METHOD INTERNAL ParseResponsePayload : DINT
VAR_INPUT
  /// Response data
  ResponseData : RobotLibraryRecvDataFB;
  /// Timestamp
  Timestamp    : SystemTime;  
END_VAR
// Table 6-77: Received CMD payload (RC to PLC) of "SwitchLanguage"
// --------------------------
// Header
// --------------------------
// Byte 00 : USINT - ParSeq | State     
// Byte 01 : SINT  - AlarmMessageSeverity    
// Byte 02 : UINT  - AlarmMessageCode HB
// Byte 03 :       - AlarmMessageCode LB
// --------------------------
// Datablock
// --------------------------
// Byte 04  : BOOL - SoftMovement
// call base implementation to parse the header from payload buffer
ResponseData.PayloadPtr := SUPER^.ParseResponsePayload(ResponseData := ResponseData, Timestamp := Timestamp);

// copy parsed header to response
_response.ParSeq               := _rspHeader.ParSeq;
_response.State                := _rspHeader.State;
_response.AlarmMessageSeverity := _rspHeader.AlarmMessageSeverity;
_response.AlarmMessageCode     := _rspHeader.AlarmMessageCode;

// Get Response.ActualLanguageCode
_response.ActualLanguageCode := ResponseData.GetString(2);

// Create logging
ParseResponsePayloadLog(ResponseData := ResponseData, Timestamp := Timestamp);
END_METHOD

METHOD INTERNAL ParseResponsePayloadLog
VAR_INPUT
  /// Response data
  ResponseData : RobotLibraryRecvDataFB;
  /// Timestamp
  Timestamp    : SystemTime;  
END_VAR
// Create log entry for Parameter start
CreateLogMessage      ( Timestamp   := Timestamp,
                        MessageType := MessageType.CMD,
                        Severity    := Severity.DEBUG,
                        MessageCode := 0,
                        MessageText := 'Parsed the following parameter(s) from response data:');
                        
// Create log entry for ActualLanguageCode
CreateLogMessagePara1 ( Timestamp   := Timestamp,
                        MessageType := MessageType.CMD,
                        Severity    := Severity.DEBUG,
                        MessageCode := 0,
                        MessageText := 'Response.ActualLanguageCode = {1}',
                        Para1       := _response.ActualLanguageCode);
END_METHOD

METHOD PROTECTED Reset : DINT
VAR_INPUT
END_VAR
Reset := SUPER^.Reset();

Done               := FALSE;
Busy               := FALSE;
CommandBuffered    := FALSE;
END_METHOD

END_FUNCTION_BLOCK

// Library/POUs/General/MC_UserLogin/MC_UserLoginFB
/// Login on RC from PLC
FUNCTION_BLOCK MC_UserLoginFB EXTENDS RobotLibraryBaseExecuteFB
// ------------------------------------------------------------------------- 
//  SRCI Robot Library                                                
// ------------------------------------------------------------------------- 
//                                                                           
//  Object:      UserLoginFB                                       
//  Author:      Thorsten Brach                                                
//  Date:        2024-06-01
//
//  Description:                                              
//   
//                                                                           
//  Copyright: 
//    (C) 2024 Thorsten Brach. All rights reserved                                                                                                                                            
//             Licensed under the LGPL-3.0 license.
//                                                                           
//  Disclaimer:                                                                           
//    This project is provided without any guarantee and can be used for   
//    private and commercial purposes. Any use is at the user’s 
//    own risk and responsibility.
//
// -------------------------------------------------------------------------
VAR_INPUT
  /// Command parameter 
  ParCmd          : UserLoginParCmd;      
END_VAR
VAR_OUTPUT
  /// Command is transferred and confirmed by the RC
  CommandBuffered : BOOL;
  /// command results
  OutCmd          : UserLoginOutCmd;     
END_VAR

VAR
  /// internal copy of command parameter 
 _parCmd          : UserLoginParCmd;
  /// command data to send
 _command         : UserLoginSendData;
  /// response data received
 _response        : UserLoginRecvData;      
END_VAR

SUPER^(AxesGroup := AxesGroup);

METHOD PROTECTED CheckFunctionSupported : BOOL
VAR_IN_OUT
  /// Robot assignment of function
  AxesGroup : AxesGroup; 
END_VAR
CheckFunctionSupported := AxesGroup.InternalData.RCSupportedFunctions.UserLogin;

IF ( NOT CheckFunctionSupported )
THEN
  // call base implementation for set error and create log entry
  SUPER^.CheckFunctionSupported(AxesGroup := AxesGroup);
END_IF
END_METHOD

METHOD PROTECTED CheckParameterChanged : BOOL
VAR_IN_OUT
  /// Robot assignment of function
  AxesGroup    : AxesGroup; 
END_VAR
// Check ParCmd Size is > 0, because MemCmp does not work correctly with size = 0
IF (SIZEOF(ParCmd) = 0) 
THEN 
  RETURN;
END_IF

// compare memory 
_parameterChanged := ( SysDepMemCmp(pData1 := ADR(ParCmd), pData2 := ADR(_parCmd), DataLen := SIZEOF(ParCmd)) <> RobotLibraryConstants.OK );

// check parameter valid ?
_parameterValid   := CheckParameterValid( AxesGroup := AxesGroup );

IF ((  _parameterChanged        )  AND 
    (  _parameterValid          )) OR
    (  _parameterUpdateInternal )  
THEN  
  // reset internal flag for send parameter update
 _parameterUpdateInternal := FALSE;
  // update internal copy of parameters 
 _parCmd := ParCmd;
  // inc parameter sequence
 _command.ParSeq := _command.ParSeq + 1;
  // update command data  
  CommandData := CreateCommandPayload(AxesGroup := AxesGroup); // ( Access via reference to rCommandFB in ACR )
  // notify active command register 
  AxesGroup.Acyclic.ActiveCommandRegister.NotifyParameterChanged := _uniqueID;
END_IF
END_METHOD

METHOD INTERNAL CreateCommandPayload : RobotLibrarySendDataFB
VAR_IN_OUT
  /// Robot assignment of function
  AxesGroup : AxesGroup; 
END_VAR
// Table 6-69: Sent CMD payload (PLC to RC) of "UserLogin"
// --------------------------
// Header
// --------------------------
// Byte 00 : UINT  - Type HB     
// Byte 01 :       - Type LB    
// Byte 02 : USINT - Reserve | ExecutionMode
// Byte 03 : USINT - ParSeq  | Priority
// --------------------------
// Datablock
// --------------------------
// Byte 04 : SINT       - Mode
// Byte 05 : SINT       - LevelID
// Byte 06 : String(50) - Password[0]
// Byte 07 :            - Password[1]
// Byte 08 :            - Password[2]
// Byte 09 :            - Password[3]
// Byte 10 :            - Password[4]
// Byte 11 :            - Password[5]
// Byte 12 :            - Password[6]
// Byte 13 :            - Password[7]
// Byte 14 :            - Password[8]
// Byte 15 :            - Password[9]
// Byte 16 :            - Password[10]
// Byte 17 :            - Password[11]
// Byte 18 :            - Password[12]
// Byte 19 :            - Password[13]
// Byte 20 :            - Password[14]
// Byte 21 :            - Password[15]
// Byte 22 :            - Password[16]
// Byte 23 :            - Password[17]
// Byte 24 :            - Password[18]
// Byte 25 :            - Password[19]
// Byte 26 :            - Password[20]
// Byte 27 :            - Password[21]
// Byte 28 :            - Password[22]
// Byte 29 :            - Password[23]
// Byte 30 :            - Password[24]
// Byte 31 :            - Password[25]
// Byte 32 :            - Password[26]
// Byte 33 :            - Password[27]
// Byte 34 :            - Password[28]
// Byte 35 :            - Password[29]
// Byte 36 :            - Password[30]
// Byte 37 :            - Password[31]
// Byte 38 :            - Password[32]
// Byte 39 :            - Password[33]
// Byte 40 :            - Password[34]
// Byte 41 :            - Password[35]
// Byte 42 :            - Password[36]
// Byte 43 :            - Password[37]
// Byte 44 :            - Password[38]
// Byte 45 :            - Password[39]
// Byte 46 :            - Password[40]
// Byte 47 :            - Password[41]
// Byte 48 :            - Password[42]
// Byte 49 :            - Password[43]
// Byte 50 :            - Password[44]
// Byte 51 :            - Password[45]
// Byte 52 :            - Password[46]
// Byte 53 :            - Password[47]
// Byte 54 :            - Password[48]
// Byte 55 :            - Password[49]
// Byte 56 : String(50) - Username[0]
// Byte 57 :            - Username[1]
// Byte 58 :            - Username[2]
// Byte 59 :            - Username[3]
// Byte 60 :            - Username[4]
// Byte 61 :            - Username[5]
// Byte 62 :            - Username[6]
// Byte 63 :            - Username[7]
// Byte 64 :            - Username[8]
// Byte 65 :            - Username[9]
// Byte 66 :            - Username[10]
// Byte 67 :            - Username[11]
// Byte 68 :            - Username[12]
// Byte 69 :            - Username[13]
// Byte 70 :            - Username[14]
// Byte 71 :            - Username[15]
// Byte 72 :            - Username[16]
// Byte 73 :            - Username[17]
// Byte 74 :            - Username[18]
// Byte 75 :            - Username[19]
// Byte 76 :            - Username[20]
// Byte 77 :            - Username[21]
// Byte 78 :            - Username[22]
// Byte 79 :            - Username[23]
// Byte 80 :            - Username[24]
// Byte 81 :            - Username[25]
// Byte 82 :            - Username[26]
// Byte 83 :            - Username[27]
// Byte 84 :            - Username[28]
// Byte 85 :            - Username[29]
// Byte 86 :            - Username[30]
// Byte 87 :            - Username[31]
// Byte 88 :            - Username[32]
// Byte 89 :            - Username[33]
// Byte 90 :            - Username[34]
// Byte 91 :            - Username[35]
// Byte 92 :            - Username[36]
// Byte 93 :            - Username[37]
// Byte 94 :            - Username[38]
// Byte 95 :            - Username[39]
// Byte 96 :            - Username[40]
// Byte 97 :            - Username[41]
// Byte 98 :            - Username[42]
// Byte 99 :            - Username[43]
// Byte 100:            - Username[44]
// Byte 101:            - Username[45]
// Byte 102:            - Username[46]
// Byte 103:            - Username[47]
// Byte 104:            - Username[48]
// Byte 105:            - Username[49]
// set command parameter 
_command.CmdTyp     :=  CmdType.UserLogin;
_command.ExecMode   :=  ExecMode;
_command.ParSeq     := _command.ParSeq;
_command.Priority   :=  Priority;

_command.Mode       := _parCmd.Mode;
_command.LevelID    := _parCmd.LevelID;
_command.Username   := _parCmd.Username;
_command.Password   := _parCmd.Password;


// copy command data to header
_cmdHeader := _command;
// call base implementation to copy header to payload buffer
CreateCommandPayload := SUPER^.CreateCommandPayload(AxesGroup := AxesGroup);

// add command.Mode
CreateCommandPayload.AddSint(_command.Mode);
// add command.LevelID
CreateCommandPayload.AddSint(_command.LevelID);
// add command.Password
CreateCommandPayload.AddString(_command.Password);
// add command.Username
CreateCommandPayload.AddString(_command.Username);

// Create logging
CreateCommandPayloadLog(AxesGroup := AxesGroup);
END_METHOD

METHOD INTERNAL CreateCommandPayloadLog 
VAR_IN_OUT
  /// Robot assignment of function
  AxesGroup : AxesGroup; 
END_VAR
// Create log entry for Parameter start
CreateLogMessage      ( Timestamp   := AxesGroup.InternalData.SystemTime,
                        MessageType := MessageType.CMD,
                        Severity    := Severity.DEBUG,
                        MessageCode := 0,
                        MessageText := 'Create command payload with the following parameter(s) :');

// Create log entry for Mode
CreateLogMessagePara1 ( Timestamp   := AxesGroup.InternalData.SystemTime,
                        MessageType := MessageType.CMD,
                        Severity    := Severity.DEBUG,
                        MessageCode := 0,
                        MessageText := 'Command.Mode = {1}',
                        Para1       :=  LOGON_MODE_TO_STRING(_command.Mode));

// Create log entry for LevelID
CreateLogMessagePara1 ( Timestamp   := AxesGroup.InternalData.SystemTime,
                        MessageType := MessageType.CMD,
                        Severity    := Severity.DEBUG,
                        MessageCode := 0,
                        MessageText := 'Command.LevelID = {1}',
                        Para1       :=  SINT_TO_STRING(_command.LevelID));

// Create log entry for Password
CreateLogMessagePara1 ( Timestamp   := AxesGroup.InternalData.SystemTime,
                        MessageType := MessageType.CMD,
                        Severity    := Severity.DEBUG,
                        MessageCode := 0,
                        MessageText := 'Command.Password = {1}',
                        Para1       :=  _command.Password);

// Create log entry for Username
CreateLogMessagePara1 ( Timestamp   := AxesGroup.InternalData.SystemTime,
                        MessageType := MessageType.CMD,
                        Severity    := Severity.DEBUG,
                        MessageCode := 0,
                        MessageText := 'Command.Username = {1}',
                        Para1       :=  _command.Username);
END_METHOD

METHOD FB_init : BOOL
VAR_INPUT
  /// if TRUE, the retain variables are initialized (warm start / cold start)
  bInitRetains : BOOL; 
  /// if TRUE, the instance afterwards gets moved into the copy code (online change)
  bInCopyCode  : BOOL;  
END_VAR
MyType := 'MC_UserLoginFB';

ExecMode := ExecutionMode.PARALLEL;
END_METHOD

METHOD PROTECTED OnCall
VAR_IN_OUT
  /// Robot assignment of function
  AxesGroup : AxesGroup; 
END_VAR
// call base implementation
SUPER^.OnCall(AxesGroup := AxesGroup);

CASE _stepCmd OF
  
  00:  IF ( _execute_R.Q )  
       THEN
         // Check function is supported and parameter are valid ?
         IF (( CheckFunctionSupported( AxesGroup := AxesGroup )) AND
             ( CheckParameterValid   ( AxesGroup := AxesGroup )))      
         THEN
           // set busy flag
           Busy := TRUE;
           // Reset command outputs
           SysDepMemSet(pDest := ADR(OutCmd), Value := 0, DataLen := SIZEOF(OutCmd));         
           // apply command parameter
          _parCmd := ParCmd;
           // init parameter sequence
          _command.ParSeq := 1;
           // create command data
           CommandData := CreateCommandPayload(AxesGroup := AxesGroup);
           // Add command to active command register
          _uniqueID := AxesGroup.Acyclic.ActiveCommandRegister.AddCmd( pCommandFB := ADR(THIS^ ));     
           // set timeout
           SetTimeout(PT := _timeoutCmd, rTimer := _timerCmd);
           // inc step counter
          _stepCmd := _stepCmd + 1; 
         END_IF
       END_IF
     

  01:  // Wait for responce received
       IF ( _responseReceived )
       THEN
         // reset response received flag
        _responseReceived := FALSE;

         CASE  _response.State 
         OF
           CmdMessageState.BUFFERED : CommandBuffered := TRUE;
           CmdMessageState.DONE     : Done            := TRUE;
           CmdMessageState.ERROR    : Error           := TRUE;
         END_CASE
                
         // Done, Aborted or Error ?
         IF (_response.State >= CmdMessageState.DONE )
         THEN
           // Reset Busy flag
           Busy := FALSE;
           // Update results
           // set timeout
           SetTimeout(PT := _timeoutCmd, rTimer := _timerCmd);
           // inc step counter
          _stepCmd := _stepCmd + 1; 
         END_IF
       END_IF


  02: IF ( NOT Execute)
      THEN
        Reset();
      END_IF     

ELSE
  // invalid step
  ErrorID := RobotLibraryEvents.ERR_INVALID_STEP;
END_CASE


// Reset FB
IF ( NOT Execute )
THEN
  Reset();
END_IF
END_METHOD

METHOD INTERNAL ParseResponsePayload : DINT
VAR_INPUT
  /// Response data
  ResponseData : RobotLibraryRecvDataFB;
  /// Timestamp
  Timestamp    : SystemTime;  
END_VAR
// Table 6-70: Received CMD payload (RC to PLC) of "UserLogin"
// --------------------------
// Header
// --------------------------
// Byte 00 : USINT - ParSeq | State     
// Byte 01 : SINT  - AlarmMessageSeverity    
// Byte 02 : UINT  - AlarmMessageCode HB
// Byte 03 :       - AlarmMessageCode LB
// --------------------------
// call base implementation to parse the header from payload buffer
ResponseData.PayloadPtr := SUPER^.ParseResponsePayload(ResponseData := ResponseData, Timestamp := Timestamp);

// copy parsed header to response
_response.ParSeq               := _rspHeader.ParSeq;
_response.State                := _rspHeader.State;
_response.AlarmMessageSeverity := _rspHeader.AlarmMessageSeverity;
_response.AlarmMessageCode     := _rspHeader.AlarmMessageCode;

// Create logging
ParseResponsePayloadLog(ResponseData := ResponseData, Timestamp := Timestamp);
END_METHOD

METHOD INTERNAL ParseResponsePayloadLog
VAR_INPUT
  /// Response data
  ResponseData : RobotLibraryRecvDataFB;
  /// Timestamp
  Timestamp    : SystemTime;  
END_VAR
// Create log entry for Parameter start
CreateLogMessage      ( Timestamp   := Timestamp,
                        MessageType := MessageType.CMD,
                        Severity    := Severity.DEBUG,
                        MessageCode := 0,
                        MessageText := 'Parsed the following parameter(s) from response data:');
                        
// Create log entry for no parameter 
CreateLogMessage      ( Timestamp   := Timestamp,
                        MessageType := MessageType.CMD,
                        Severity    := Severity.DEBUG,
                        MessageCode := 0,
                        MessageText := 'This command has no parameter to parse...');
END_METHOD

METHOD PROTECTED Reset : DINT
VAR_INPUT
END_VAR
Reset := SUPER^.Reset();

Done               := FALSE;
Busy               := FALSE;
CommandBuffered    := FALSE;
END_METHOD

END_FUNCTION_BLOCK

// Library/POUs/Read/MC_ReadActualPosition/MC_ReadActualPositionFB
/// Read the actual position – TCP: X…RZ + config/Turn, … Joint: (J1…E6)
FUNCTION_BLOCK MC_ReadActualPositionFB EXTENDS RobotLibraryBaseExecuteFB
// ------------------------------------------------------------------------- 
//  SRCI Robot Library                                                
// ------------------------------------------------------------------------- 
//                                                                           
//  Object:      ReadActualPositionFB                                       
//  Author:      Thorsten Brach                                                
//  Date:        2024-06-01
//
//  Description:                                              
//   
//                                                                           
//  Copyright: 
//    (C) 2024 Thorsten Brach. All rights reserved                                                                                                                                            
//             Licensed under the LGPL-3.0 license.
//                                                                           
//  Disclaimer:                                                                           
//    This project is provided without any guarantee and can be used for   
//    private and commercial purposes. Any use is at the user’s 
//    own risk and responsibility.
//
// -------------------------------------------------------------------------
VAR_INPUT
  /// Processing mode - For more information see chapter 5.6.4.5.
  ProcessingMode     : ProcessingMode;
  /// Defines the target sequence in which the command will be executed
  SequenceFlag       : SequenceFlag;  
  /// command parameter 
  ParCmd             : ReadActualPositionParCmd;
END_VAR

VAR_OUTPUT
  /// TRUE, while the following outputs return valid values
  /// • ActualCartesianPosition
  /// • ToolNoReturn
  /// • FrameNoReturn
  /// • ActualJointPosition
  Valid              : BOOL;
  /// Command is transferred and confirmed by the RC
  CommandBuffered    : BOOL;  
  /// The command was aborted by another command.
  CommandAborted     : BOOL;
  /// TRUE, while command is interrupted during execution and can be continued.
  CommandInterrupted : BOOL;
  /// Receiving of input parameter values has been acknowledged by RC
  ParameterAccepted  : BOOL;
  /// command outputs
  OutCmd             : ReadActualPositionOutCmd;       
END_VAR

VAR
  /// internal copy of command parameter 
 _parCmd             : ReadActualPositionParCmd;
  /// command data to send
 _command            : ReadActualPositionSendData;
  /// response data received
 _response           : ReadActualPositionRecvData;      
END_VAR

SUPER^(AxesGroup := AxesGroup);

METHOD PROTECTED CheckFunctionSupported : BOOL
VAR_IN_OUT
  /// Robot assignment of function
  AxesGroup : AxesGroup; 
END_VAR
CheckFunctionSupported := AxesGroup.InternalData.RCSupportedFunctions.ReadActualPosition;

IF ( NOT CheckFunctionSupported )
THEN
  // call base implementation for set error and create log entry
  SUPER^.CheckFunctionSupported(AxesGroup := AxesGroup);
END_IF
END_METHOD

METHOD PROTECTED CheckParameterChanged : BOOL
VAR_IN_OUT
  /// Robot assignment of function
  AxesGroup    : AxesGroup; 
END_VAR
// Check ParCmd Size is > 0, because MemCmp does not work correctly with size = 0
IF (SIZEOF(ParCmd) = 0) 
THEN 
  RETURN;
END_IF

// compare memory 
_parameterChanged := ( SysDepMemCmp(pData1 := ADR(ParCmd), pData2 := ADR(_parCmd), DataLen := SIZEOF(ParCmd)) <> RobotLibraryConstants.OK );

// check parameter valid ?
_parameterValid   := CheckParameterValid( AxesGroup := AxesGroup );

IF ((  _parameterChanged        )  AND 
    (  _parameterValid          )) OR
    (  _parameterUpdateInternal )  
THEN  
  // reset internal flag for send parameter update
 _parameterUpdateInternal := FALSE;
  // update internal copy of parameters 
 _parCmd := ParCmd;
  // inc parameter sequence
 _command.ParSeq := _command.ParSeq + 1;
  // update command data  
  CommandData := CreateCommandPayload(AxesGroup := AxesGroup); // ( Access via reference to rCommandFB in ACR )
  // notify active command register 
  AxesGroup.Acyclic.ActiveCommandRegister.NotifyParameterChanged := _uniqueID;
  // Reset parameter accepted flag
  ParameterAccepted := FALSE;  
END_IF
END_METHOD

METHOD INTERNAL CreateCommandPayload : RobotLibrarySendDataFB
VAR_IN_OUT
  /// Robot assignment of function
  AxesGroup : AxesGroup; 
END_VAR
// Table 6-38: Sent CMD payload (PLC to RC) of "ReadActualPosition"
// --------------------------
// Header
// --------------------------
// Byte 00 : UINT  - Type HB     
// Byte 01 :       - Type LB    
// Byte 02 : USINT - Reserve | ExecutionMode
// Byte 03 : USINT - ParSeq  | Priority
// --------------------------
// Datablock
// --------------------------
// Byte 04 : SINT  EmitterID[0];
// Byte 05 : SINT  EmitterID[1];
// Byte 06 : SINT  EmitterID[2];
// Byte 07 : SINT  EmitterID[3];
// Byte 08 : SINT  ListenerID;
// Byte 09 : BYTE  Reserved;
// Byte 10 : USINT ToolNo
// Byte 11 : USINT FrameNo
// --------------------------
// set command parameter 
_command.CmdTyp       :=  CmdType.ReadActualPosition;
_command.ExecMode     :=  ExecMode;
_command.ParSeq       := _command.ParSeq;
_command.Priority     :=  Priority;
_command.EmitterID[0] := 0;
_command.EmitterID[1] := 0;
_command.EmitterID[2] := 0;
_command.EmitterID[3] := 0;
_command.Reserve      := 0;
_command.ListenerID   := _parCmd.ListenerID;
_command.ToolNo       := INT_TO_USINT(_parCmd.ToolNo);
_command.FrameNo      := INT_TO_USINT(_parCmd.FrameNo);


// copy command data to header
_cmdHeader := _command;
// call base implementation to copy header to payload buffer
CreateCommandPayload := SUPER^.CreateCommandPayload(AxesGroup := AxesGroup);

// add command.EmitterID[0]
CreateCommandPayload.AddSint(_command.EmitterID[0]);
// add command.EmitterID[1]
CreateCommandPayload.AddSint(_command.EmitterID[1]);
// add command.EmitterID[2]
CreateCommandPayload.AddSint(_command.EmitterID[2]);
// add command.EmitterID[3]
CreateCommandPayload.AddSint(_command.EmitterID[3]);
// add command.ListenerID
CreateCommandPayload.AddSint(_command.ListenerID);
// add command.Reserve
CreateCommandPayload.AddByte(_command.Reserve);
// add command.Index[0]
CreateCommandPayload.AddUsint(_command.ToolNo);
// add command.Index[1]
CreateCommandPayload.AddUsint(_command.FrameNo);

// Create logging
CreateCommandPayloadLog(AxesGroup := AxesGroup);
END_METHOD

METHOD INTERNAL CreateCommandPayloadLog
VAR_IN_OUT
  /// Robot assignment of function
  AxesGroup : AxesGroup; 
END_VAR
VAR 
  /// internal index for loops
 _idx : DINT;
END_VAR
// Create log entry for Parameter start
CreateLogMessage      ( Timestamp   := AxesGroup.InternalData.SystemTime,
                        MessageType := MessageType.CMD,
                        Severity    := Severity.DEBUG,
                        MessageCode := 0,
                        MessageText := 'Create command payload with the following parameter(s) :');
  
// Create log entry for EmitterID[x]
FOR _idx := 0 TO 3
DO
  CreateLogMessagePara2 ( Timestamp   := AxesGroup.InternalData.SystemTime,
                          MessageType := MessageType.CMD,
                          Severity    := Severity.DEBUG,
                          MessageCode := 0,
                          MessageText := 'Command.EmitterID[{2}] = {1}',
                          Para1       :=  SINT_TO_STRING(_command.EmitterID[_idx]),
                          Para2       :=  DINT_TO_STRING(_idx));
END_FOR

// Create log entry for ListenerID
CreateLogMessagePara1 ( Timestamp   := AxesGroup.InternalData.SystemTime,
                        MessageType := MessageType.CMD,
                        Severity    := Severity.DEBUG,
                        MessageCode := 0,
                        MessageText := 'Command.ListenerID = {1}',
                        Para1       :=  SINT_TO_STRING(_command.ListenerID));
                        
// Create log entry for Reserve
CreateLogMessagePara1 ( Timestamp   := AxesGroup.InternalData.SystemTime,
                        MessageType := MessageType.CMD,
                        Severity    := Severity.DEBUG,
                        MessageCode := 0,
                        MessageText := 'Command.Reserve = {1}',
                        Para1       :=  BYTE_TO_STRING(_command.Reserve));

// Create log entry for ToolNo
CreateLogMessagePara1 ( Timestamp   := AxesGroup.InternalData.SystemTime,
                        MessageType := MessageType.CMD,
                        Severity    := Severity.DEBUG,
                        MessageCode := 0,
                        MessageText := 'Command.ToolNo = {1}',
                        Para1       :=  USINT_TO_STRING(_command.ToolNo));

// Create log entry for FrameNo
CreateLogMessagePara1 ( Timestamp   := AxesGroup.InternalData.SystemTime,
                        MessageType := MessageType.CMD,
                        Severity    := Severity.DEBUG,
                        MessageCode := 0,
                        MessageText := 'Command.FrameNo = {1}',
                        Para1       :=  USINT_TO_STRING(_command.FrameNo));
END_METHOD

METHOD FB_init : BOOL
VAR_INPUT
  /// if TRUE, the retain variables are initialized (warm start / cold start)
  bInitRetains : BOOL; 
  /// if TRUE, the instance afterwards gets moved into the copy code (online change)
  bInCopyCode  : BOOL;  
END_VAR
MyType := 'MC_ReadActualPositionFB';

ExecMode := ExecutionMode.PARALLEL;
END_METHOD

METHOD PROTECTED OnCall
VAR_IN_OUT
  /// Robot assignment of function
  AxesGroup : AxesGroup; 
END_VAR
// call base implementation
SUPER^.OnCall(AxesGroup := AxesGroup);

CASE _stepCmd OF
  
  00:  IF ( _execute_R.Q )  
       THEN
         // Check function is supported and parameter are valid ?
         IF (( CheckFunctionSupported( AxesGroup := AxesGroup )) AND
             ( CheckParameterValid   ( AxesGroup := AxesGroup )))      
         THEN
           // set busy flag
           Busy := TRUE;
           // Reset command outputs
           SysDepMemSet(pDest := ADR(OutCmd), Value := 0, DataLen := SIZEOF(OutCmd));         
           // apply command parameter
          _parCmd := ParCmd;
           // init parameter sequence
          _command.ParSeq := 1;
           // create command data
           CommandData := CreateCommandPayload(AxesGroup := AxesGroup);
           // Add command to active command register
          _uniqueID := AxesGroup.Acyclic.ActiveCommandRegister.AddCmd( pCommandFB := ADR(THIS^ ));     
           // set timeout
           SetTimeout(PT := _timeoutCmd, rTimer := _timerCmd);
           // inc step counter
          _stepCmd := _stepCmd + 1;
         END_IF 
       END_IF
     

  01:  // Wait for responce received
       IF ( _responseReceived )
       THEN
         // reset response received flag
        _responseReceived := FALSE;

         CASE  _response.State 
         OF
           CmdMessageState.BUFFERED    : CommandBuffered    := TRUE;
           CmdMessageState.ACTIVE      : ParameterAccepted  := TRUE;           
           CmdMessageState.INTERRUPTED : CommandInterrupted := TRUE;           
           CmdMessageState.DONE        : Done               := TRUE;
           CmdMessageState.ABORTED     : CommandAborted     := TRUE;
           CmdMessageState.ERROR       : Error              := TRUE;
         END_CASE
                
         // Done, Aborted or Error ?
         IF (_response.State >= CmdMessageState.DONE )
         THEN
           // Reset Busy flag
           Busy := FALSE;
           // Update results
           OutCmd.OriginID                := _response.OriginID;
           OutCmd.InvocationCounter       := _response.InvocationCounter;
           OutCmd.ToolNoReturn            := _response.ToolNoReturn;
           OutCmd.FrameNoReturn           := _response.FrameNoReturn;
           OutCmd.ActualCartesianPosition := _response.ActualCartesianPosition;
           OutCmd.ActualJointPosition     := _response.ActualJointPosition;
           // set timeout
           SetTimeout(PT := _timeoutCmd, rTimer := _timerCmd);
           // inc step counter
          _stepCmd := _stepCmd + 1; 
         END_IF
       END_IF


  02: IF ( NOT Execute)
      THEN
        Reset();
      END_IF     
      
ELSE
  // invalid step
  ErrorID := RobotLibraryEvents.ERR_INVALID_STEP;
END_CASE


// Reset FB
IF ( NOT Execute )
THEN
  Reset();
END_IF
END_METHOD

METHOD INTERNAL ParseResponsePayload : DINT
VAR_INPUT
  /// Response data
  ResponseData : RobotLibraryRecvDataFB;
  /// Timestamp
  Timestamp    : SystemTime;  
END_VAR
// Table 6-39: Received CMD payload (RC to PLC) of "ReadActualPosition"
// --------------------------
// Header
// --------------------------
// Byte 00 : USINT   - ParSeq | State     
// Byte 01 : SINT    - AlarmMessageSeverity    
// Byte 02 : UINT    - AlarmMessageCode HB
// Byte 03 :         - AlarmMessageCode LB
// --------------------------
// Datablock
// --------------------------
// Byte 04 : USINT   - InvocationCounter;
// Byte 05 : SINT    - Reserved;
// Byte 06 : INT     - OriginID HW HB;
// Byte 07 :         - OriginID HW LB;
// Byte 08 : USINT   - ToolNoReturn;
// Byte 09 : USINT   - FrameNoReturn;
// Byte 10 : REAL    - ActualCartesianPosition.X HW HB;
// Byte 11 :         - ActualCartesianPosition.X HW LB;
// Byte 12 :         - ActualCartesianPosition.X LW HB;
// Byte 13 :         - ActualCartesianPosition.X LW LB;
// Byte 14 : REAL    - ActualCartesianPosition.Y HW HB;
// Byte 15 :         - ActualCartesianPosition.Y HW LB;
// Byte 16 :         - ActualCartesianPosition.Y LW HB;
// Byte 17 :         - ActualCartesianPosition.Y LW LB;
// Byte 18 : REAL    - ActualCartesianPosition.Z HW HB;
// Byte 19 :         - ActualCartesianPosition.Z HW LB;
// Byte 20 :         - ActualCartesianPosition.Z LW HB;
// Byte 21 :         - ActualCartesianPosition.Z LW LB;
// Byte 22 : REAL    - ActualCartesianPosition.RX HW HB;
// Byte 23 :         - ActualCartesianPosition.RX HW LB;
// Byte 24 :         - ActualCartesianPosition.RX LW HB;
// Byte 25 :         - ActualCartesianPosition.RX LW LB;
// Byte 26 : REAL    - ActualCartesianPosition.RY HW HB;
// Byte 27 :         - ActualCartesianPosition.RY HW LB;
// Byte 28 :         - ActualCartesianPosition.RY LW HB;
// Byte 29 :         - ActualCartesianPosition.RY LW LB;
// Byte 30 : REAL    - ActualCartesianPosition.RZ HW HB;
// Byte 31 :         - ActualCartesianPosition.RZ HW LB;
// Byte 32 :         - ActualCartesianPosition.RZ LW HB;
// Byte 33 :         - ActualCartesianPosition.RZ LW LB;
// Byte 34 : BYTE    - W E S;
// Byte 35 : BYTE    - Reserved;
// Byte 36 : BYTE    - ActualCartesianPosition.TurnNumber[0];
// Byte 37 : BYTE    - ActualCartesianPosition.TurnNumber[1];
// Byte 38 : BYTE    - ActualCartesianPosition.TurnNumber[2];
// Byte 39 : BYTE    - ActualCartesianPosition.TurnNumber[3];
// Byte 40 : REAL    - ActualJointPosition.J1 HW HB;
// Byte 41 :         - ActualJointPosition.J1 HW LB;
// Byte 42 :         - ActualJointPosition.J1 LW HB;
// Byte 43 :         - ActualJointPosition.J1 LW LB;
// Byte 44 : REAL    - ActualJointPosition.J2 HW HB;
// Byte 45 :         - ActualJointPosition.J2 HW LB;
// Byte 46 :         - ActualJointPosition.J2 LW HB;
// Byte 47 :         - ActualJointPosition.J2 LW LB;
// Byte 48 : REAL    - ActualJointPosition.J3 HW HB;
// Byte 49 :         - ActualJointPosition.J3 HW LB;
// Byte 50 :         - ActualJointPosition.J3 LW HB;
// Byte 51 :         - ActualJointPosition.J3 LW LB;
// Byte 52 : REAL    - ActualJointPosition.J4 HW HB;
// Byte 53 :         - ActualJointPosition.J4 HW LB;
// Byte 54 :         - ActualJointPosition.J4 LW HB;
// Byte 55 :         - ActualJointPosition.J4 LW LB;
// Byte 56 : REAL    - ActualJointPosition.J5 HW HB;
// Byte 57 :         - ActualJointPosition.J5 HW LB;
// Byte 58 :         - ActualJointPosition.J5 LW HB;
// Byte 59 :         - ActualJointPosition.J5 LW LB;
// Byte 60 : REAL    - ActualJointPosition.J6 HW HB;
// Byte 61 :         - ActualJointPosition.J6 HW LB;
// Byte 62 :         - ActualJointPosition.J6 LW HB;
// Byte 63 :         - ActualJointPosition.J6 LW LB;
// Byte 64 : REAL    - ActualCartesianPosition.E1 HW HB;
// Byte 65 :         - ActualCartesianPosition.E1 HW LB;
// Byte 66 :         - ActualCartesianPosition.E1 LW HB;
// Byte 67 :         - ActualCartesianPosition.E1 LW LB;
// Byte 68 : REAL    - ActualCartesianPosition.E2 HW HB;
// Byte 69 :         - ActualCartesianPosition.E2 HW LB;
// Byte 70 :         - ActualCartesianPosition.E2 LW HB;
// Byte 71 :         - ActualCartesianPosition.E2 LW LB;
// Byte 72 : REAL    - ActualCartesianPosition.E3 HW HB;
// Byte 73 :         - ActualCartesianPosition.E3 HW LB;
// Byte 74 :         - ActualCartesianPosition.E3 LW HB;
// Byte 75 :         - ActualCartesianPosition.E3 LW LB;
// Byte 76 : REAL    - ActualCartesianPosition.E4 HW HB;
// Byte 77 :         - ActualCartesianPosition.E4 HW LB;
// Byte 78 :         - ActualCartesianPosition.E4 LW HB;
// Byte 79 :         - ActualCartesianPosition.E4 LW LB;
// Byte 80 : REAL    - ActualCartesianPosition.E5 HW HB;
// Byte 81 :         - ActualCartesianPosition.E5 HW LB;
// Byte 82 :         - ActualCartesianPosition.E5 LW HB;
// Byte 83 :         - ActualCartesianPosition.E5 LW LB;
// Byte 84 : REAL    - ActualCartesianPosition.E6 HW HB;
// Byte 85 :         - ActualCartesianPosition.E6 HW LB;
// Byte 86 :         - ActualCartesianPosition.E6 LW HB;
// Byte 87 :         - ActualCartesianPosition.E6 LW LB;
// Byte 88 : REAL    - ActualJointPosition.E1 HW HB;
// Byte 89 :         - ActualJointPosition.E1 HW LB;
// Byte 90 :         - ActualJointPosition.E1 LW HB;
// Byte 91 :         - ActualJointPosition.E1 LW LB;
// Byte 92 : REAL    - ActualJointPosition.E2 HW HB;
// Byte 93 :         - ActualJointPosition.E2 HW LB;
// Byte 94 :         - ActualJointPosition.E2 LW HB;
// Byte 95 :         - ActualJointPosition.E2 LW LB;
// Byte 96 : REAL    - ActualJointPosition.E3 HW HB;
// Byte 97 :         - ActualJointPosition.E3 HW LB;
// Byte 98 :         - ActualJointPosition.E3 LW HB;
// Byte 99 :         - ActualJointPosition.E3 LW LB;
// Byte 100: REAL    - ActualJointPosition.E4 HW HB;
// Byte 101:         - ActualJointPosition.E4 HW LB;
// Byte 102:         - ActualJointPosition.E4 LW HB;
// Byte 103:         - ActualJointPosition.E4 LW LB;
// Byte 104: REAL    - ActualJointPosition.E5 HW HB;
// Byte 105:         - ActualJointPosition.E5 HW LB;
// Byte 106:         - ActualJointPosition.E5 LW HB;
// Byte 107:         - ActualJointPosition.E5 LW LB;
// Byte 108: REAL    - ActualJointPosition.E6 HW HB;
// Byte 109:         - ActualJointPosition.E6 HW LB;
// Byte 110:         - ActualJointPosition.E6 LW HB;
// Byte 111:         - ActualJointPosition.E6 LW LB;
// --------------------------
// call base implementation to parse the header from payload buffer
ResponseData.PayloadPtr := SUPER^.ParseResponsePayload(ResponseData := ResponseData, Timestamp := Timestamp);

// copy parsed header to response
_response.ParSeq               := _rspHeader.ParSeq;
_response.State                := _rspHeader.State;
_response.AlarmMessageSeverity := _rspHeader.AlarmMessageSeverity;
_response.AlarmMessageCode     := _rspHeader.AlarmMessageCode;

// Get Response.InvocationCounter
_response.InvocationCounter := ResponseData.GetUsint();
// Get Response.Reserve
_response.Reserve := ResponseData.GetSint();
// Get Response.OriginID
_response.OriginID := ResponseData.GetInt();

// Get Response.ToolNoReturn
_response.ToolNoReturn := ResponseData.GetUsint();
// Get Response.FrameNoReturn
_response.FrameNoReturn := ResponseData.GetUsint();
// Get Response.ActualCartesianPosition.X
_response.ActualCartesianPosition.X := ResponseData.GetReal();
// Get Response.ActualCartesianPosition.Y
_response.ActualCartesianPosition.Y := ResponseData.GetReal();
// Get Response.ActualCartesianPosition.Z
_response.ActualCartesianPosition.Z := ResponseData.GetReal();
// Get Response.ActualCartesianPosition.Rx
_response.ActualCartesianPosition.Rx := ResponseData.GetReal();
// Get Response.ActualCartesianPosition.Ry
_response.ActualCartesianPosition.Ry := ResponseData.GetReal();
// Get Response.ActualCartesianPosition.Rz
_response.ActualCartesianPosition.Rz := ResponseData.GetReal();
// Get Response.ActualCartesianPosition.Config
_response.ActualCartesianPosition.Config := ResponseData.GetArmConfig();
// Get Response.ActualCartesianPosition.TurnNumber
_response.ActualCartesianPosition.TurnNumber := ResponseData.GetTurnNumbers();
// Get Response.ActualCartesianPosition.E1
_response.ActualCartesianPosition.E1 := ResponseData.GetReal();
// Get Response.ActualJointPosition.J1
_response.ActualJointPosition.J1 := ResponseData.GetReal();
// Get Response.ActualJointPosition.J2
_response.ActualJointPosition.J2 := ResponseData.GetReal();
// Get Response.ActualJointPosition.J3
_response.ActualJointPosition.J3 := ResponseData.GetReal();
// Get Response.ActualJointPosition.J4
_response.ActualJointPosition.J4 := ResponseData.GetReal();
// Get Response.ActualJointPosition.J5
_response.ActualJointPosition.J5 := ResponseData.GetReal();
// Get Response.ActualJointPosition.J6
_response.ActualJointPosition.J6 := ResponseData.GetReal();
// Get Response.ActualCartesianPosition.E2
_response.ActualCartesianPosition.E2 := ResponseData.GetReal();
// Get Response.ActualCartesianPosition.E3
_response.ActualCartesianPosition.E3 := ResponseData.GetReal();
// Get Response.ActualCartesianPosition.E4
_response.ActualCartesianPosition.E4 := ResponseData.GetReal();
// Get Response.ActualCartesianPosition.E5
_response.ActualCartesianPosition.E5 := ResponseData.GetReal();
// Get Response.ActualCartesianPosition.E6
_response.ActualCartesianPosition.E6 := ResponseData.GetReal();
// Get Response.ActualJointPosition.E1
_response.ActualJointPosition.E1 := ResponseData.GetReal();
// Get Response.ActualJointPosition.E2
_response.ActualJointPosition.E2 := ResponseData.GetReal();
// Get Response.ActualJointPosition.E3
_response.ActualJointPosition.E3 := ResponseData.GetReal();
// Get Response.ActualJointPosition.E4
_response.ActualJointPosition.E4 := ResponseData.GetReal();
// Get Response.ActualJointPosition.E5
_response.ActualJointPosition.E5 := ResponseData.GetReal();
// Get Response.ActualJointPosition.E6
_response.ActualJointPosition.E6 := ResponseData.GetReal();

// Create logging
ParseResponsePayloadLog(ResponseData := ResponseData, Timestamp := Timestamp);
END_METHOD

METHOD INTERNAL ParseResponsePayloadLog
VAR_INPUT
  /// Response data
  ResponseData : RobotLibraryRecvDataFB;
  /// Timestamp
  Timestamp    : SystemTime;  
END_VAR
// Create log entry for Parameter start
CreateLogMessage      ( Timestamp   := Timestamp,
                        MessageType := MessageType.CMD,
                        Severity    := Severity.DEBUG,
                        MessageCode := 0,
                        MessageText := 'Parsed the following parameter(s) from response data:');

// Create log entry for InvocationCounter
CreateLogMessagePara1 ( Timestamp   := Timestamp,
                        MessageType := MessageType.CMD,
                        Severity    := Severity.DEBUG,
                        MessageCode := 0,
                        MessageText := 'Response.InvocationCounter = {1}',
                        Para1       :=  USINT_TO_STRING(_response.InvocationCounter));

// Create log entry for Reserve
CreateLogMessagePara1 ( Timestamp   := Timestamp,
                        MessageType := MessageType.CMD,
                        Severity    := Severity.DEBUG,
                        MessageCode := 0,
                        MessageText := 'Response.Reserve = {1}',
                        Para1       :=  SINT_TO_STRING(_response.Reserve));

// Create log entry for OriginID
CreateLogMessagePara1 ( Timestamp   := Timestamp,
                        MessageType := MessageType.CMD,
                        Severity    := Severity.DEBUG,
                        MessageCode := 0,
                        MessageText := 'Response.OriginID = {1}',
                        Para1       :=  INT_TO_STRING(_response.OriginID));

// Create log entry for ToolNoReturn
CreateLogMessagePara1 ( Timestamp   := Timestamp,
                        MessageType := MessageType.CMD,
                        Severity    := Severity.DEBUG,
                        MessageCode := 0,
                        MessageText := 'Response.ToolNoReturn = {1}',
                        Para1       :=  INT_TO_STRING(_response.ToolNoReturn));

// Create log entry for FrameNoReturn
CreateLogMessagePara1 ( Timestamp   := Timestamp,
                        MessageType := MessageType.CMD,
                        Severity    := Severity.DEBUG,
                        MessageCode := 0,
                        MessageText := 'Response.FrameNoReturn = {1}',
                        Para1       :=  INT_TO_STRING(_response.FrameNoReturn));

// Create log entry for ActualCartesianPosition.X
CreateLogMessagePara1 ( Timestamp   := Timestamp,
                        MessageType := MessageType.CMD,
                        Severity    := Severity.DEBUG,
                        MessageCode := 0,
                        MessageText := 'Response.ActualCartesianPosition.X = {1}',
                        Para1       :=  REAL_TO_STRING(_response.ActualCartesianPosition.X));

// Create log entry for ActualCartesianPosition.Y
CreateLogMessagePara1 ( Timestamp   := Timestamp,
                        MessageType := MessageType.CMD,
                        Severity    := Severity.DEBUG,
                        MessageCode := 0,
                        MessageText := 'Response.ActualCartesianPosition.Y = {1}',
                        Para1       :=  REAL_TO_STRING(_response.ActualCartesianPosition.Y));

// Create log entry for ActualCartesianPosition.Z
CreateLogMessagePara1 ( Timestamp   := Timestamp,
                        MessageType := MessageType.CMD,
                        Severity    := Severity.DEBUG,
                        MessageCode := 0,
                        MessageText := 'Response.ActualCartesianPosition.Z = {1}',
                        Para1       :=  REAL_TO_STRING(_response.ActualCartesianPosition.Z));

// Create log entry for ActualCartesianPosition.Rx
CreateLogMessagePara1 ( Timestamp   := Timestamp,
                        MessageType := MessageType.CMD,
                        Severity    := Severity.DEBUG,
                        MessageCode := 0,
                        MessageText := 'Response.ActualCartesianPosition.Rx = {1}',
                        Para1       :=  REAL_TO_STRING(_response.ActualCartesianPosition.Rx));
                        
// Create log entry for ActualCartesianPosition.Ry
CreateLogMessagePara1 ( Timestamp   := Timestamp,
                        MessageType := MessageType.CMD,
                        Severity    := Severity.DEBUG,
                        MessageCode := 0,
                        MessageText := 'Response.ActualCartesianPosition.Ry = {1}',
                        Para1       :=  REAL_TO_STRING(_response.ActualCartesianPosition.Ry));

// Create log entry for ActualCartesianPosition.Rz
CreateLogMessagePara1 ( Timestamp   := Timestamp,
                        MessageType := MessageType.CMD,
                        Severity    := Severity.DEBUG,
                        MessageCode := 0,
                        MessageText := 'Response.ActualCartesianPosition.Rz = {1}',
                        Para1       :=  REAL_TO_STRING(_response.ActualCartesianPosition.Rz));


// Create log entry for ActualCartesianPosition.Config
CreateLogMessagePara1 ( Timestamp   := Timestamp,
                        MessageType := MessageType.CMD,
                        Severity    := Severity.DEBUG,
                        MessageCode := 0,
                        MessageText := 'Response.ActualCartesianPosition.Config = {1}',
                        Para1       :=  ARM_CONFIG_TO_STRING(_response.ActualCartesianPosition.Config));

// Create log entry for ActualCartesianPosition.TurnNumber.J1Turns
CreateLogMessagePara1 ( Timestamp   := Timestamp,
                        MessageType := MessageType.CMD,
                        Severity    := Severity.DEBUG,
                        MessageCode := 0,
                        MessageText := 'Response.ActualCartesianPosition.TurnNumber.J1Turns = {1}',
                        Para1       :=  SINT_TO_STRING(_response.ActualCartesianPosition.TurnNumber.J1Turns));

// Create log entry for ActualCartesianPosition.TurnNumber.J2Turns
CreateLogMessagePara1 ( Timestamp   := Timestamp,
                        MessageType := MessageType.CMD,
                        Severity    := Severity.DEBUG,
                        MessageCode := 0,
                        MessageText := 'Response.ActualCartesianPosition.TurnNumber.J2Turns = {1}',
                        Para1       :=  SINT_TO_STRING(_response.ActualCartesianPosition.TurnNumber.J2Turns));

// Create log entry for ActualCartesianPosition.TurnNumber.J3Turns
CreateLogMessagePara1 ( Timestamp   := Timestamp,
                        MessageType := MessageType.CMD,
                        Severity    := Severity.DEBUG,
                        MessageCode := 0,
                        MessageText := 'Response.ActualCartesianPosition.TurnNumber.J3Turns = {1}',
                        Para1       :=  SINT_TO_STRING(_response.ActualCartesianPosition.TurnNumber.J3Turns));

// Create log entry for ActualCartesianPosition.TurnNumber.J4Turns
CreateLogMessagePara1 ( Timestamp   := Timestamp,
                        MessageType := MessageType.CMD,
                        Severity    := Severity.DEBUG,
                        MessageCode := 0,
                        MessageText := 'Response.ActualCartesianPosition.TurnNumber.J4Turns = {1}',
                        Para1       :=  SINT_TO_STRING(_response.ActualCartesianPosition.TurnNumber.J4Turns));

// Create log entry for ActualCartesianPosition.TurnNumber.J5Turns
CreateLogMessagePara1 ( Timestamp   := Timestamp,
                        MessageType := MessageType.CMD,
                        Severity    := Severity.DEBUG,
                        MessageCode := 0,
                        MessageText := 'Response.ActualCartesianPosition.TurnNumber.J5Turns = {1}',
                        Para1       :=  SINT_TO_STRING(_response.ActualCartesianPosition.TurnNumber.J5Turns));

// Create log entry for ActualCartesianPosition.TurnNumber.J6Turns
CreateLogMessagePara1 ( Timestamp   := Timestamp,
                        MessageType := MessageType.CMD,
                        Severity    := Severity.DEBUG,
                        MessageCode := 0,
                        MessageText := 'Response.ActualCartesianPosition.TurnNumber.J6Turns = {1}',
                        Para1       :=  SINT_TO_STRING(_response.ActualCartesianPosition.TurnNumber.J6Turns));

// Create log entry for ActualCartesianPosition.TurnNumber.E1Turns
CreateLogMessagePara1 ( Timestamp   := Timestamp,
                        MessageType := MessageType.CMD,
                        Severity    := Severity.DEBUG,
                        MessageCode := 0,
                        MessageText := 'Response.ActualCartesianPosition.TurnNumber.E1Turns = {1}',
                        Para1       :=  SINT_TO_STRING(_response.ActualCartesianPosition.TurnNumber.E1Turns));

// Create log entry for ActualCartesianPosition.E1
CreateLogMessagePara1 ( Timestamp   := Timestamp,
                        MessageType := MessageType.CMD,
                        Severity    := Severity.DEBUG,
                        MessageCode := 0,
                        MessageText := 'Response.ActualCartesianPosition.E1 = {1}',
                        Para1       :=  REAL_TO_STRING(_response.ActualCartesianPosition.E1));

// Create log entry for ActualJointPosition.J1
CreateLogMessagePara1 ( Timestamp   := Timestamp,
                        MessageType := MessageType.CMD,
                        Severity    := Severity.DEBUG,
                        MessageCode := 0,
                        MessageText := 'Response.ActualJointPosition.J1 = {1}',
                        Para1       :=  REAL_TO_STRING(_response.ActualJointPosition.J1));

// Create log entry for ActualJointPosition.J2
CreateLogMessagePara1 ( Timestamp   := Timestamp,
                        MessageType := MessageType.CMD,
                        Severity    := Severity.DEBUG,
                        MessageCode := 0,
                        MessageText := 'Response.ActualJointPosition.J2 = {1}',
                        Para1       :=  REAL_TO_STRING(_response.ActualJointPosition.J2));

// Create log entry for ActualJointPosition.J3
CreateLogMessagePara1 ( Timestamp   := Timestamp,
                        MessageType := MessageType.CMD,
                        Severity    := Severity.DEBUG,
                        MessageCode := 0,
                        MessageText := 'Response.ActualJointPosition.J3 = {1}',
                        Para1       :=  REAL_TO_STRING(_response.ActualJointPosition.J3));

// Create log entry for ActualJointPosition.J4
CreateLogMessagePara1 ( Timestamp   := Timestamp,
                        MessageType := MessageType.CMD,
                        Severity    := Severity.DEBUG,
                        MessageCode := 0,
                        MessageText := 'Response.ActualJointPosition.J4 = {1}',
                        Para1       :=  REAL_TO_STRING(_response.ActualJointPosition.J4));

// Create log entry for ActualJointPosition.J5
CreateLogMessagePara1 ( Timestamp   := Timestamp,
                        MessageType := MessageType.CMD,
                        Severity    := Severity.DEBUG,
                        MessageCode := 0,
                        MessageText := 'Response.ActualJointPosition.J5 = {1}',
                        Para1       :=  REAL_TO_STRING(_response.ActualJointPosition.J5));

// Create log entry for ActualJointPosition.J6
CreateLogMessagePara1 ( Timestamp   := Timestamp,
                        MessageType := MessageType.CMD,
                        Severity    := Severity.DEBUG,
                        MessageCode := 0,
                        MessageText := 'Response.ActualJointPosition.J6 = {1}',
                        Para1       :=  REAL_TO_STRING(_response.ActualJointPosition.J6));

// Create log entry for ActualJointPosition.E1
CreateLogMessagePara1 ( Timestamp   := Timestamp,
                        MessageType := MessageType.CMD,
                        Severity    := Severity.DEBUG,
                        MessageCode := 0,
                        MessageText := 'Response.ActualJointPosition.E1 = {1}',
                        Para1       :=  REAL_TO_STRING(_response.ActualJointPosition.E1));

// Create log entry for ActualCartesianPosition.E2
CreateLogMessagePara1 ( Timestamp   := Timestamp,
                        MessageType := MessageType.CMD,
                        Severity    := Severity.DEBUG,
                        MessageCode := 0,
                        MessageText := 'Response.ActualCartesianPosition.E2 = {1}',
                        Para1       :=  REAL_TO_STRING(_response.ActualCartesianPosition.E2));
                        
// Create log entry for ActualCartesianPosition.E3
CreateLogMessagePara1 ( Timestamp   := Timestamp,
                        MessageType := MessageType.CMD,
                        Severity    := Severity.DEBUG,
                        MessageCode := 0,
                        MessageText := 'Response.ActualCartesianPosition.E3 = {1}',
                        Para1       :=  REAL_TO_STRING(_response.ActualCartesianPosition.E3));

// Create log entry for ActualCartesianPosition.E4
CreateLogMessagePara1 ( Timestamp   := Timestamp,
                        MessageType := MessageType.CMD,
                        Severity    := Severity.DEBUG,
                        MessageCode := 0,
                        MessageText := 'Response.ActualCartesianPosition.E4 = {1}',
                        Para1       :=  REAL_TO_STRING(_response.ActualCartesianPosition.E4));

// Create log entry for ActualCartesianPosition.E5
CreateLogMessagePara1 ( Timestamp   := Timestamp,
                        MessageType := MessageType.CMD,
                        Severity    := Severity.DEBUG,
                        MessageCode := 0,
                        MessageText := 'Response.ActualCartesianPosition.E5 = {1}',
                        Para1       :=  REAL_TO_STRING(_response.ActualCartesianPosition.E5));

// Create log entry for ActualCartesianPosition.E6
CreateLogMessagePara1 ( Timestamp   := Timestamp,
                        MessageType := MessageType.CMD,
                        Severity    := Severity.DEBUG,
                        MessageCode := 0,
                        MessageText := 'Response.ActualCartesianPosition.E6 = {1}',
                        Para1       :=  REAL_TO_STRING(_response.ActualCartesianPosition.E6));           

// Create log entry for ActualJointPosition.E2
CreateLogMessagePara1 ( Timestamp   := Timestamp,
                        MessageType := MessageType.CMD,
                        Severity    := Severity.DEBUG,
                        MessageCode := 0,
                        MessageText := 'Response.ActualJointPosition.E2 = {1}',
                        Para1       :=  REAL_TO_STRING(_response.ActualJointPosition.E2));

// Create log entry for ActualJointPosition.E3
CreateLogMessagePara1 ( Timestamp   := Timestamp,
                        MessageType := MessageType.CMD,
                        Severity    := Severity.DEBUG,
                        MessageCode := 0,
                        MessageText := 'Response.ActualJointPosition.E3 = {1}',
                        Para1       :=  REAL_TO_STRING(_response.ActualJointPosition.E3));
                        
// Create log entry for ActualJointPosition.E4
CreateLogMessagePara1 ( Timestamp   := Timestamp,
                        MessageType := MessageType.CMD,
                        Severity    := Severity.DEBUG,
                        MessageCode := 0,
                        MessageText := 'Response.ActualJointPosition.E4 = {1}',
                        Para1       :=  REAL_TO_STRING(_response.ActualJointPosition.E4));

// Create log entry for ActualJointPosition.E5
CreateLogMessagePara1 ( Timestamp   := Timestamp,
                        MessageType := MessageType.CMD,
                        Severity    := Severity.DEBUG,
                        MessageCode := 0,
                        MessageText := 'Response.ActualJointPosition.E5 = {1}',
                        Para1       :=  REAL_TO_STRING(_response.ActualJointPosition.E5));
                        
// Create log entry for ActualJointPosition.E6
CreateLogMessagePara1 ( Timestamp   := Timestamp,
                        MessageType := MessageType.CMD,
                        Severity    := Severity.DEBUG,
                        MessageCode := 0,
                        MessageText := 'Response.ActualJointPosition.E6 = {1}',
                        Para1       :=  REAL_TO_STRING(_response.ActualJointPosition.E6));
END_METHOD

METHOD PROTECTED Reset : DINT
VAR_INPUT
END_VAR
Reset := SUPER^.Reset();

Done               := FALSE;
Busy               := FALSE;
Valid              := FALSE;
ParameterAccepted  := FALSE;
CommandBuffered    := FALSE;
CommandAborted     := FALSE;
CommandInterrupted := FALSE;
END_METHOD

END_FUNCTION_BLOCK

// Library/POUs/Read/MC_ReadActualPositionCyclic/MC_ReadActualPositionCyclicFB
/// Read the actual position cyclically
FUNCTION_BLOCK MC_ReadActualPositionCyclicFB EXTENDS RobotLibraryBaseEnableFB
// ------------------------------------------------------------------------- 
//  SRCI Robot Library                                                
// ------------------------------------------------------------------------- 
//                                                                           
//  Object:      ReadActualPositionCyclicFB                                       
//  Author:      Thorsten Brach                                                
//  Date:        2024-06-01
//
//  Description:                                              
//   
//                                                                           
//  Copyright: 
//    (C) 2024 Thorsten Brach. All rights reserved                                                                                                                                            
//             Licensed under the LGPL-3.0 license.
//                                                                           
//  Disclaimer:                                                                           
//    This project is provided without any guarantee and can be used for   
//    private and commercial purposes. Any use is at the user’s 
//    own risk and responsibility.
//
// -------------------------------------------------------------------------
VAR_INPUT
  /// command parameter 
  ParCmd   : ReadActualPositionCyclicParCmd;
END_VAR

VAR_OUTPUT
  /// command outputs
  OutCmd   : ReadActualPositionCyclicOutCmd;       
END_VAR

VAR
  /// internal copy of command parameter 
 _parCmd   : ReadActualPositionCyclicParCmd;
END_VAR

SUPER^(AxesGroup := AxesGroup);

METHOD PROTECTED CheckFunctionSupported : BOOL
VAR_IN_OUT
  /// Robot assignment of function
  AxesGroup : AxesGroup; 
END_VAR
CheckFunctionSupported := AxesGroup.InternalData.RCSupportedFunctions.ReadActualPositionCyclic;

IF ( NOT CheckFunctionSupported )
THEN
  // call base implementation for set error and create log entry
  SUPER^.CheckFunctionSupported(AxesGroup := AxesGroup);
END_IF
END_METHOD

METHOD PROTECTED CheckParameterChanged : BOOL
VAR_IN_OUT
  /// Robot assignment of function
  AxesGroup : AxesGroup; 
END_VAR
// Check ParCmd Size is > 0, because MemCmp does not work correctly with size = 0
IF (SIZEOF(ParCmd) = 0) 
THEN 
  RETURN;
END_IF

// compare memory 
_parameterChanged := ( SysDepMemCmp(pData1 := ADR(ParCmd), pData2 := ADR(_parCmd), DataLen := SIZEOF(ParCmd)) <> RobotLibraryConstants.OK );

// check parameter valid ?
_parameterValid   := CheckParameterValid( AxesGroup := AxesGroup );

IF ((  _parameterChanged        )  AND 
    (  _parameterValid          )) OR
    (  _parameterUpdateInternal )  
THEN  
  // reset internal flag for send parameter update
 _parameterUpdateInternal := FALSE;
  // Set busy flag
  Busy := TRUE;
  // reset enable flag
  Enabled := FALSE;
  // update internal copy of parameters 
 _parCmd := ParCmd;
  // update tool number 
  AxesGroup.Cyclic.PlcToRob.ToolNo  := _parCmd.ToolNo;
  // update frame number 
  AxesGroup.Cyclic.PlcToRob.FrameNo := _parCmd.FrameNo;
  // Create logging
  CreateCommandParameterLog(AxesGroup := AxesGroup);
END_IF
END_METHOD

METHOD PROTECTED CheckParameterValid : BOOL
VAR_IN_OUT
  /// Robot assignment of function
  AxesGroup : AxesGroup; 
END_VAR
CheckParameterValid := TRUE;

// Check ParCmd are valid ? 
IF (( ParCmd.ReadCartesianPosition    ) AND ( NOT AxesGroup.CyclicOptional.RobToPlc.CartesianPosition   .Active) OR
    ( ParCmd.ReadCartesianPositionExt ) AND ( NOT AxesGroup.CyclicOptional.RobToPlc.CartesianPositionExt.Active) OR
    ( ParCmd.ReadJointPosition        ) AND ( NOT AxesGroup.CyclicOptional.RobToPlc.JointPosition       .Active) OR
    ( ParCmd.ReadJointPositionExt     ) AND ( NOT AxesGroup.CyclicOptional.RobToPlc.JointPositionExt    .Active))
THEN
  CheckParameterValid := FALSE;
END_IF
END_METHOD

METHOD INTERNAL CreateCommandParameterLog
VAR_IN_OUT
  /// Robot assignment of function
  AxesGroup : AxesGroup; 
END_VAR
// Create log entry for Parameter start
CreateLogMessage      ( Timestamp   := AxesGroup.InternalData.SystemTime,
                        MessageType := MessageType.CMD,
                        Severity    := Severity.DEBUG,
                        MessageCode := 0,
                        MessageText := 'Update position with the following parameter(s) :');
                        
// Create log entry for _parCmd.ReadCartesianPosition
CreateLogMessagePara1 ( Timestamp   := AxesGroup.InternalData.SystemTime,
                        MessageType := MessageType.CMD,
                        Severity    := Severity.DEBUG,
                        MessageCode := 0,
                        MessageText := '_parCmd.ReadCartesianPosition = {1}',
                        Para1       :=  BOOL_TO_STRING(_parCmd.ReadCartesianPosition));

// Create log entry for _parCmd.ReadCartesianPositionExt
CreateLogMessagePara1 ( Timestamp   := AxesGroup.InternalData.SystemTime,
                        MessageType := MessageType.CMD,
                        Severity    := Severity.DEBUG,
                        MessageCode := 0,
                        MessageText := '_parCmd.ReadCartesianPositionExt = {1}',
                        Para1       :=  BOOL_TO_STRING(_parCmd.ReadCartesianPositionExt));

// Create log entry for _parCmd.ToolNo
CreateLogMessagePara1 ( Timestamp   := AxesGroup.InternalData.SystemTime,
                        MessageType := MessageType.CMD,
                        Severity    := Severity.DEBUG,
                        MessageCode := 0,
                        MessageText := '_parCmd.ToolNo = {1}',
                        Para1       :=  INT_TO_STRING(_parCmd.ToolNo));

// Create log entry for _parCmd.FrameNo
CreateLogMessagePara1 ( Timestamp   := AxesGroup.InternalData.SystemTime,
                        MessageType := MessageType.CMD,
                        Severity    := Severity.DEBUG,
                        MessageCode := 0,
                        MessageText := '_parCmd.FrameNo = {1}',
                        Para1       :=  INT_TO_STRING(_parCmd.FrameNo));

// Create log entry for _parCmd.ReadJointPosition
CreateLogMessagePara1 ( Timestamp   := AxesGroup.InternalData.SystemTime,
                        MessageType := MessageType.CMD,
                        Severity    := Severity.DEBUG,
                        MessageCode := 0,
                        MessageText := '_parCmd.ReadJointPosition = {1}',
                        Para1       :=  BOOL_TO_STRING(_parCmd.ReadJointPosition));

// Create log entry for _parCmd.ReadJointPositionExt
CreateLogMessagePara1 ( Timestamp   := AxesGroup.InternalData.SystemTime,
                        MessageType := MessageType.CMD,
                        Severity    := Severity.DEBUG,
                        MessageCode := 0,
                        MessageText := '_parCmd.ReadJointPositionExt = {1}',
                        Para1       :=  BOOL_TO_STRING(_parCmd.ReadJointPositionExt));
END_METHOD

METHOD FB_init : BOOL
VAR_INPUT
  /// if TRUE, the retain variables are initialized (warm start / cold start)
  bInitRetains : BOOL; 
  /// if TRUE, the instance afterwards gets moved into the copy code (online change)
  bInCopyCode  : BOOL;  
END_VAR
MyType := 'MC_ReadActualPositionCyclicFB';
END_METHOD

METHOD PROTECTED OnCall
VAR_IN_OUT
  /// Robot assignment of function
  AxesGroup : AxesGroup; 
END_VAR
SUPER^.OnCall(AxesGroup := AxesGroup);

CASE _stepCmd OF
  
  00:  IF ( _enable_R.Q ) 
       THEN
         // reset the rising edge
        _enable_R();       
         // reset the falling edge
        _enable_F();
        
         // Check function is supported and parameter are valid ?
         IF (( CheckFunctionSupported( AxesGroup := AxesGroup )) AND
             ( CheckParameterValid   ( AxesGroup := AxesGroup )))      
         THEN
           // set busy flag
           Busy := TRUE;
           // Reset command outputs
           SysDepMemSet(pDest := ADR(OutCmd), Value := 0, DataLen := SIZEOF(OutCmd));         
           // apply command parameter
          _parCmd := ParCmd;
           // set parameter
           AxesGroup.Cyclic.PlcToRob.ToolNo  := _parCmd.ToolNo;
           AxesGroup.Cyclic.PlcToRob.FrameNo := _parCmd.FrameNo;   
           // Create logging
           CreateCommandParameterLog(AxesGroup := AxesGroup);  
           // set timeout
           SetTimeout(PT := _timeoutCmd, rTimer := _timerCmd);
           // inc step counter
          _stepCmd := _stepCmd + 1; 
         END_IF 
       END_IF
     

  01:  // Wait for FrameNo and ToolNo set
       IF ((  AxesGroup.CyclicOptional.RobToPlc.CartesianPosition.CoordinateSystem.FrameNo = _parCmd.FrameNo )  AND
           (  AxesGroup.CyclicOptional.RobToPlc.CartesianPosition.CoordinateSystem.ToolNo  = _parCmd.ToolNo  )) OR
           ( _parCmd.ReadCartesianPosition                                                 = FALSE           ) 
       THEN
         // busy 
         Busy := FALSE;
         // reset busy flag
         Enabled := TRUE;          
         // Reset command outputs
         SysDepMemSet(pDest := ADR(OutCmd), Value := 0, DataLen := SIZEOF(OutCmd));         
         // set ToolNo and FrameNo
         OutCmd.CurrentCoordinateSystem.FrameNo := AxesGroup.CyclicOptional.RobToPlc.CartesianPosition.CoordinateSystem.FrameNo;
         OutCmd.CurrentCoordinateSystem.ToolNo  := AxesGroup.CyclicOptional.RobToPlc.CartesianPosition.CoordinateSystem.ToolNo;
         
         // Set cartesian position
         IF ( _parCmd.ReadCartesianPosition )  
         THEN
            OutCmd.ReadingCartesianPosition     := TRUE;
            OutCmd.CartesianPosition.X          := OutCmd.CartesianPositionShort.X          := AxesGroup.CyclicOptional.RobToPlc.CartesianPosition.X;
            OutCmd.CartesianPosition.Y          := OutCmd.CartesianPositionShort.Y          := AxesGroup.CyclicOptional.RobToPlc.CartesianPosition.Y;         
            OutCmd.CartesianPosition.Z          := OutCmd.CartesianPositionShort.Z          := AxesGroup.CyclicOptional.RobToPlc.CartesianPosition.Z;
            OutCmd.CartesianPosition.Rx         := OutCmd.CartesianPositionShort.Rx         := AxesGroup.CyclicOptional.RobToPlc.CartesianPosition.Rx;
            OutCmd.CartesianPosition.Ry         := OutCmd.CartesianPositionShort.Ry         := AxesGroup.CyclicOptional.RobToPlc.CartesianPosition.Ry;
            OutCmd.CartesianPosition.Rz         := OutCmd.CartesianPositionShort.Rz         := AxesGroup.CyclicOptional.RobToPlc.CartesianPosition.Rz;
            OutCmd.CartesianPosition.Config     := OutCmd.CartesianPositionShort.Config     := AxesGroup.CyclicOptional.RobToPlc.CartesianPosition.Config;
            OutCmd.CartesianPosition.TurnNumber := OutCmd.CartesianPositionShort.TurnNumber := AxesGroup.CyclicOptional.RobToPlc.CartesianPosition.TurnNumber;            
            OutCmd.CartesianPosition.E1         := OutCmd.CartesianPositionShort.E1         := AxesGroup.CyclicOptional.RobToPlc.CartesianPosition.E1;
         END_IF
         
         // Set extended cartesian position
         IF ( _parCmd.ReadCartesianPositionExt )  
         THEN
            OutCmd.ReadingCartesianPositionExt  := TRUE;
            OutCmd.CartesianPosition.E2         := OutCmd.CartesianPositionExt.E2           := AxesGroup.CyclicOptional.RobToPlc.CartesianPositionExt.E2;
            OutCmd.CartesianPosition.E3         := OutCmd.CartesianPositionExt.E3           := AxesGroup.CyclicOptional.RobToPlc.CartesianPositionExt.E3;
            OutCmd.CartesianPosition.E4         := OutCmd.CartesianPositionExt.E4           := AxesGroup.CyclicOptional.RobToPlc.CartesianPositionExt.E4;
            OutCmd.CartesianPosition.E5         := OutCmd.CartesianPositionExt.E5           := AxesGroup.CyclicOptional.RobToPlc.CartesianPositionExt.E5;
            OutCmd.CartesianPosition.E6         := OutCmd.CartesianPositionExt.E6           := AxesGroup.CyclicOptional.RobToPlc.CartesianPositionExt.E6;    
         END_IF      

         // Set joint position
         IF ( _parCmd.ReadJointPosition )  
         THEN
            OutCmd.ReadingJointPosition         := TRUE;         
            OutCmd.JointPosition.J1             := OutCmd.JointPositionShort.J1             := AxesGroup.CyclicOptional.RobToPlc.JointPosition.J1;
            OutCmd.JointPosition.J2             := OutCmd.JointPositionShort.J2             := AxesGroup.CyclicOptional.RobToPlc.JointPosition.J2;
            OutCmd.JointPosition.J3             := OutCmd.JointPositionShort.J3             := AxesGroup.CyclicOptional.RobToPlc.JointPosition.J3;
            OutCmd.JointPosition.J4             := OutCmd.JointPositionShort.J4             := AxesGroup.CyclicOptional.RobToPlc.JointPosition.J4;
            OutCmd.JointPosition.J5             := OutCmd.JointPositionShort.J5             := AxesGroup.CyclicOptional.RobToPlc.JointPosition.J5;
            OutCmd.JointPosition.J6             := OutCmd.JointPositionShort.J6             := AxesGroup.CyclicOptional.RobToPlc.JointPosition.J6;    
         END_IF    
  
         // Set extended joint position
         IF ( _parCmd.ReadJointPositionExt )  
         THEN         
            OutCmd.ReadingCartesianPositionExt  := TRUE;         
            OutCmd.JointPosition.E2             := OutCmd.JointPositionExt.E2               := AxesGroup.CyclicOptional.RobToPlc.JointPositionExt.E2;
            OutCmd.JointPosition.E3             := OutCmd.JointPositionExt.E3               := AxesGroup.CyclicOptional.RobToPlc.JointPositionExt.E3;
            OutCmd.JointPosition.E4             := OutCmd.JointPositionExt.E4               := AxesGroup.CyclicOptional.RobToPlc.JointPositionExt.E4;
            OutCmd.JointPosition.E5             := OutCmd.JointPositionExt.E5               := AxesGroup.CyclicOptional.RobToPlc.JointPositionExt.E5;
            OutCmd.JointPosition.E6             := OutCmd.JointPositionExt.E6               := AxesGroup.CyclicOptional.RobToPlc.JointPositionExt.E6;    
         END_IF
       END_IF
       
       IF ( NOT Enable)
       THEN
         // reset the rising edge
        _enable_R();       
         // reset the falling edge
        _enable_F();       
         // set timeout
         SetTimeout(PT := _timeoutCmd, rTimer := _timerCmd);
         // inc step counter
        _stepCmd := _stepCmd + 1; 
       END_IF


  02:  IF (NOT Enable)
       THEN
         Reset();  
       END_IF

ELSE
  // invalid step
  ErrorID := RobotLibraryEvents.ERR_INVALID_STEP;
END_CASE



// Reset FB
IF (( _enable_R.Q ) OR
    ( _enable_F.Q ))
THEN
  Reset();
END_IF
END_METHOD

METHOD PROTECTED Reset : DINT
VAR_INPUT
END_VAR
Reset := SUPER^.Reset();

// Reset command outputs
SysDepMemSet(pDest := ADR(OutCmd), Value := 0, DataLen := SIZEOF(OutCmd));
END_METHOD

END_FUNCTION_BLOCK

// Library/POUs/Read/MC_ReadActualTCPVelocity/MC_ReadActualTCPVelocityFB
/// Read actual TCP velocity
FUNCTION_BLOCK MC_ReadActualTCPVelocityFB EXTENDS RobotLibraryBaseExecuteFB
// ------------------------------------------------------------------------- 
//  SRCI Robot Library                                                
// ------------------------------------------------------------------------- 
//                                                                           
//  Object:      ReadActualTCPVelocityFB                                       
//  Author:      Thorsten Brach                                                
//  Date:        2024-06-01
//
//  Description:                                              
//   
//                                                                           
//  Copyright: 
//    (C) 2024 Thorsten Brach. All rights reserved                                                                                                                                            
//             Licensed under the LGPL-3.0 license.
//                                                                           
//  Disclaimer:                                                                           
//    This project is provided without any guarantee and can be used for   
//    private and commercial purposes. Any use is at the user’s 
//    own risk and responsibility.
//
// -------------------------------------------------------------------------
VAR_INPUT
  /// Processing mode
  ProcessingMode     : ProcessingMode;
  /// Defines the target sequence in which the command will be executed 
  ///  For more information about the differentiation of sequences see chapter 5.5.3.4
  SequenceFlag       : SequenceFlag;
  /// command parameter 
  ParCmd             : ReadActualTCPVelocityParCmd;  
END_VAR

VAR_OUTPUT
  /// TRUE, while the following outputs return valid values:
  /// • ActualTCPVelocity
  /// • ToolNoReturn
  /// • FrameNoReturn
  Valid              : BOOL;
  /// The command was aborted by another command.
  CommandAborted     : BOOL;
  /// Command is transferred and confirmed by the RC
  CommandBuffered    : BOOL;
  /// TRUE, while command is interrupted during execution and can be continued
  CommandInterrupted : BOOL;
  /// Receiving of input parameter values has been acknowledged by RC
  ParameterAccepted  : BOOL;
  /// command outputs
  OutCmd             : ReadActualTCPVelocityOutCmd;       
END_VAR

VAR
  /// internal copy of command parameter 
 _parCmd             : ReadActualTCPVelocityParCmd;
  /// command data to send
 _command            : ReadActualTCPVelocitySendData;
  /// response data received
 _response           : ReadActualTCPVelocityRecvData;      
END_VAR

SUPER^(AxesGroup := AxesGroup);

METHOD PROTECTED CheckFunctionSupported : BOOL
VAR_IN_OUT
  /// Robot assignment of function
  AxesGroup : AxesGroup; 
END_VAR
CheckFunctionSupported := AxesGroup.InternalData.RCSupportedFunctions.ReadActualTCPVelocity;

IF ( NOT CheckFunctionSupported )
THEN
  // call base implementation for set error and create log entry
  SUPER^.CheckFunctionSupported(AxesGroup := AxesGroup);
END_IF
END_METHOD

METHOD PROTECTED CheckParameterChanged : BOOL
VAR_IN_OUT
  /// Robot assignment of function
  AxesGroup    : AxesGroup; 
END_VAR
// Check ParCmd Size is > 0, because MemCmp does not work correctly with size = 0
IF (SIZEOF(ParCmd) = 0) 
THEN 
  RETURN;
END_IF

// compare memory 
_parameterChanged := ( SysDepMemCmp(pData1 := ADR(ParCmd), pData2 := ADR(_parCmd), DataLen := SIZEOF(ParCmd)) <> RobotLibraryConstants.OK );

// check parameter valid ?
_parameterValid   := CheckParameterValid( AxesGroup := AxesGroup );

IF ((  _parameterChanged        )  AND 
    (  _parameterValid          )) OR
    (  _parameterUpdateInternal )  
THEN  
  // reset internal flag for send parameter update
 _parameterUpdateInternal := FALSE;
  // update internal copy of parameters 
 _parCmd := ParCmd;
  // inc parameter sequence
 _command.ParSeq := _command.ParSeq + 1;
  // update command data  
  CommandData := CreateCommandPayload(AxesGroup := AxesGroup); // ( Access via reference to rCommandFB in ACR )
  // notify active command register 
  AxesGroup.Acyclic.ActiveCommandRegister.NotifyParameterChanged := _uniqueID;
  // Reset parameter accepted flag
  ParameterAccepted := FALSE;  
END_IF
END_METHOD

METHOD INTERNAL CreateCommandPayload : RobotLibrarySendDataFB
VAR_IN_OUT
  /// Robot assignment of function
  AxesGroup : AxesGroup; 
END_VAR
// Table 6-63: Sent CMD payload (PLC to RC) of "ReadActualTCPVelocity"
// --------------------------
// Header
// --------------------------
// Byte 00 : UINT  - Type HB     
// Byte 01 :       - Type LB    
// Byte 02 : USINT - Reserve | ExecutionMode
// Byte 03 : USINT - ParSeq  | Priority
// --------------------------
// Datablock
// --------------------------
// Byte 04 : USINT - ToolNo
// Byte 05 : USINT - FrameNo
// --------------------------
// set command parameter 
_command.CmdTyp                    :=  CmdType.ReadActualTCPVelocity;
_command.ExecMode                  :=  ExecMode;
_command.ParSeq                    := _command.ParSeq;
_command.Priority                  :=  Priority;
_command.ToolNo                    := _parCmd.ToolNo;
_command.FrameNo                   := _parCmd.FrameNo;


// copy command data to header
_cmdHeader := _command;
// call base implementation to copy header to payload buffer
CreateCommandPayload := SUPER^.CreateCommandPayload(AxesGroup := AxesGroup);

// add command.ToolNo
CreateCommandPayload.AddUsint(_command.ToolNo);
// add command.FrameNo
CreateCommandPayload.AddUsint(_command.FrameNo);

// Create logging
CreateCommandPayloadLog(AxesGroup := AxesGroup);
END_METHOD

METHOD INTERNAL CreateCommandPayloadLog
VAR_IN_OUT
  /// Robot assignment of function
  AxesGroup : AxesGroup; 
END_VAR

// Byte 04 : USINT - ToolNo
// Byte 05 : USINT - FrameNo
// Create log entry for Parameter start
CreateLogMessage      ( Timestamp   := AxesGroup.InternalData.SystemTime,
                        MessageType := MessageType.CMD,
                        Severity    := Severity.DEBUG,
                        MessageCode := 0,
                        MessageText := 'Create command payload with the following parameter(s) :');

// Create log entry for ToolNo
CreateLogMessagePara1 ( Timestamp   := AxesGroup.InternalData.SystemTime,
                        MessageType := MessageType.CMD,
                        Severity    := Severity.DEBUG,
                        MessageCode := 0,
                        MessageText := 'Command.ToolNo = {1}',
                        Para1       :=  USINT_TO_STRING(_command.ToolNo));

// Create log entry for FrameNo
CreateLogMessagePara1 ( Timestamp   := AxesGroup.InternalData.SystemTime,
                        MessageType := MessageType.CMD,
                        Severity    := Severity.DEBUG,
                        MessageCode := 0,
                        MessageText := 'Command.FrameNo = {1}',
                        Para1       :=  USINT_TO_STRING(_command.FrameNo));
END_METHOD

METHOD FB_init : BOOL
VAR_INPUT
  /// if TRUE, the retain variables are initialized (warm start / cold start)
  bInitRetains : BOOL; 
  /// if TRUE, the instance afterwards gets moved into the copy code (online change)
  bInCopyCode  : BOOL;  
END_VAR
MyType := 'MC_ReadActualTCPVelocityFB';

ExecMode := ExecutionMode.PARALLEL;
END_METHOD

METHOD PROTECTED OnCall
VAR_IN_OUT
  /// Robot assignment of function
  AxesGroup : AxesGroup; 
END_VAR
// call base implementation
SUPER^.OnCall(AxesGroup := AxesGroup);

CASE _stepCmd OF
  
  00:  IF ( _execute_R.Q )  
       THEN
         // Check function is supported and parameter are valid ?
         IF (( CheckFunctionSupported( AxesGroup := AxesGroup )) AND
             ( CheckParameterValid   ( AxesGroup := AxesGroup )))      
         THEN
           // set busy flag
           Busy := TRUE;
           // Reset command outputs
           SysDepMemSet(pDest := ADR(OutCmd), Value := 0, DataLen := SIZEOF(OutCmd));         
           // apply command parameter
          _parCmd := ParCmd;
           // init parameter sequence
          _command.ParSeq := 1;
           // create command data
           CommandData := CreateCommandPayload(AxesGroup := AxesGroup);
           // Add command to active command register
          _uniqueID := AxesGroup.Acyclic.ActiveCommandRegister.AddCmd( pCommandFB := ADR(THIS^ ));     
           // set timeout
           SetTimeout(PT := _timeoutCmd, rTimer := _timerCmd);
           // inc step counter
          _stepCmd := _stepCmd + 1; 
         END_IF
       END_IF
     

  01:  // Wait for responce received
       IF ( _responseReceived )
       THEN
         // reset response received flag
        _responseReceived := FALSE;

         CASE  _response.State 
         OF
           CmdMessageState.BUFFERED    : CommandBuffered    := TRUE;
           CmdMessageState.ACTIVE      : ParameterAccepted  := TRUE;
           CmdMessageState.INTERRUPTED : CommandInterrupted := TRUE;           
           CmdMessageState.DONE        : Done               := TRUE;           
           CmdMessageState.ABORTED     : CommandAborted     := TRUE;
           CmdMessageState.ERROR       : Error              := TRUE;
         END_CASE
                
         // Done, Aborted or Error ?
         IF (_response.State >= CmdMessageState.DONE )
         THEN
           // Reset Busy flag
           Busy := FALSE;
           // Update results
           OutCmd.ToolNoReturn      := _response.ToolNoReturn;
           OutCmd.FrameNoReturn     := _response.FrameNoReturn;
           OutCmd.ActualTCPVelocity := _response.ActualTCPVelocity;

           // set timeout
           SetTimeout(PT := _timeoutCmd, rTimer := _timerCmd);
           // inc step counter
          _stepCmd := _stepCmd + 1; 
         END_IF
       END_IF


  02: IF ( NOT Execute)
      THEN
        Reset();
      END_IF     

ELSE
  // invalid step
  ErrorID := RobotLibraryEvents.ERR_INVALID_STEP;
END_CASE


// Reset FB
IF ( NOT Execute )
THEN
  Reset();
END_IF
END_METHOD

METHOD INTERNAL ParseResponsePayload : DINT
VAR_INPUT
  /// Response data
  ResponseData : RobotLibraryRecvDataFB;
  /// Timestamp
  Timestamp    : SystemTime;  
END_VAR
// Table 6-64: Received CMD payload (RC to PLC) of " ReadActualTCPVelocity "
// --------------------------
// Header
// --------------------------
// Byte 00 : USINT   - ParSeq | State     
// Byte 01 : SINT    - AlarmMessageSeverity    
// Byte 02 : UINT    - AlarmMessageCode HB
// Byte 03 :         - AlarmMessageCode LB
// --------------------------
// Datablock
// --------------------------
// Byte 04 : USINT   - ToolNoReturn
// Byte 05 : USINT   - FrameNoReturn
// Byte 06 : REAL    - ActualTCPVelocity HW HB
// Byte 07 :           ActualTCPVelocity HW LB
// Byte 08 :           ActualTCPVelocity LW HB
// Byte 09 :           ActualTCPVelocity LW LB
// --------------------------
// call base implementation to parse the header from payload buffer
ResponseData.PayloadPtr := SUPER^.ParseResponsePayload(ResponseData := ResponseData, Timestamp := Timestamp);

// copy parsed header to response
_response.ParSeq               := _rspHeader.ParSeq;
_response.State                := _rspHeader.State;
_response.AlarmMessageSeverity := _rspHeader.AlarmMessageSeverity;
_response.AlarmMessageCode     := _rspHeader.AlarmMessageCode;

// Get Response.ToolNoReturn
_response.ToolNoReturn := ResponseData.GetUsint();
// Get Response.FrameNoReturn
_response.FrameNoReturn := ResponseData.GetUsint();
// Get Response.ActualTCPVelocity
_response.ActualTCPVelocity := ResponseData.GetReal();

// Create logging
ParseResponsePayloadLog(ResponseData := ResponseData, Timestamp := Timestamp);
END_METHOD

METHOD INTERNAL ParseResponsePayloadLog
VAR_INPUT
  /// Response data
  ResponseData : RobotLibraryRecvDataFB;
  /// Timestamp
  Timestamp    : SystemTime;  
END_VAR
// Create log entry for Parameter start
CreateLogMessage      ( Timestamp   := Timestamp,
                        MessageType := MessageType.CMD,
                        Severity    := Severity.DEBUG,
                        MessageCode := 0,
                        MessageText := 'Parsed the following parameter(s) from response data:');
            
// Create log entry for ToolNoReturn
CreateLogMessagePara1 ( Timestamp   := Timestamp,
                        MessageType := MessageType.CMD,
                        Severity    := Severity.DEBUG,
                        MessageCode := 0,
                        MessageText := 'Response.ToolNoReturn = {1}',
                        Para1       :=  USINT_TO_STRING(_response.ToolNoReturn));

// Create log entry for FrameNoReturn
CreateLogMessagePara1 ( Timestamp   := Timestamp,
                        MessageType := MessageType.CMD,
                        Severity    := Severity.DEBUG,
                        MessageCode := 0,
                        MessageText := 'Response.FrameNoReturn = {1}',
                        Para1       :=  USINT_TO_STRING(_response.FrameNoReturn));

// Create log entry for ActualTCPVelocity
CreateLogMessagePara1 ( Timestamp   := Timestamp,
                        MessageType := MessageType.CMD,
                        Severity    := Severity.DEBUG,
                        MessageCode := 0,
                        MessageText := 'Response.ActualTCPVelocity = {1}',
                        Para1       :=  REAL_TO_STRING(_response.ActualTCPVelocity));
END_METHOD

METHOD PROTECTED Reset : DINT
VAR_INPUT
END_VAR
Reset := SUPER^.Reset();

Done               := FALSE;
Busy               := FALSE;
Valid              := FALSE;
ParameterAccepted  := FALSE;
CommandBuffered    := FALSE;
CommandAborted     := FALSE;
CommandInterrupted := FALSE;
END_METHOD

END_FUNCTION_BLOCK

// Library/POUs/Read/MC_ReadAnalogInput/MC_ReadAnalogInputFB
/// Read analog input of RC
FUNCTION_BLOCK MC_ReadAnalogInputFB EXTENDS RobotLibraryBaseExecuteFB
// ------------------------------------------------------------------------- 
//  SRCI Robot Library                                                
// ------------------------------------------------------------------------- 
//                                                                           
//  Object:      ReadAnalogInputFB                                       
//  Author:      Thorsten Brach                                                
//  Date:        2024-06-01
//
//  Description:                                              
//   
//                                                                           
//  Copyright: 
//    (C) 2024 Thorsten Brach. All rights reserved                                                                                                                                            
//             Licensed under the LGPL-3.0 license.
//                                                                           
//  Disclaimer:                                                                           
//    This project is provided without any guarantee and can be used for   
//    private and commercial purposes. Any use is at the user’s 
//    own risk and responsibility.
//
// -------------------------------------------------------------------------
VAR_INPUT
  /// Processing Mode
  ProcessingMode     : ProcessingMode;
  /// Defines the target sequence in which the command will be executed
  SequenceFlag       : SequenceFlag;
  /// command parameter 
  ParCmd             : ReadAnalogInputParCmd;
END_VAR
VAR_OUTPUT
  /// TRUE, while the following outputs return valid values:
  /// • Values
  Valid              : BOOL; 
  /// Command is transferred and confirmed by the RC
  CommandBuffered    : BOOL;
  /// The command was aborted by another command.
  CommandAborted     : BOOL;
  /// TRUE, while command is interrupted during execution and can be continued
  CommandInterrupted : BOOL;
  /// Receiving of input parameter values has been acknowledged by RC
  ParameterAccepted  : BOOL;
  /// command outputs
  OutCmd             : ReadAnalogInputOutCmd;       
END_VAR

VAR
  /// internal copy of command parameter 
 _parCmd             : ReadAnalogInputParCmd;
  /// command data to send
 _command            : ReadAnalogInputSendData;
  /// response data received
 _response           : ReadAnalogInputRecvData;      
END_VAR

SUPER^(AxesGroup := AxesGroup);

METHOD PROTECTED CheckFunctionSupported : BOOL
VAR_IN_OUT
  /// Robot assignment of function
  AxesGroup : AxesGroup; 
END_VAR
CheckFunctionSupported := AxesGroup.InternalData.RCSupportedFunctions.ReadAnalogInput;

IF ( NOT CheckFunctionSupported )
THEN
  // call base implementation for set error and create log entry
  SUPER^.CheckFunctionSupported(AxesGroup := AxesGroup);
END_IF
END_METHOD

METHOD PROTECTED CheckParameterChanged : BOOL
VAR_IN_OUT
  /// Robot assignment of function
  AxesGroup    : AxesGroup; 
END_VAR
// Check ParCmd Size is > 0, because MemCmp does not work correctly with size = 0
IF (SIZEOF(ParCmd) = 0) 
THEN 
  RETURN;
END_IF

// compare memory 
_parameterChanged := ( SysDepMemCmp(pData1 := ADR(ParCmd), pData2 := ADR(_parCmd), DataLen := SIZEOF(ParCmd)) <> RobotLibraryConstants.OK );

// check parameter valid ?
_parameterValid   := CheckParameterValid( AxesGroup := AxesGroup );

IF ((  _parameterChanged        )  AND 
    (  _parameterValid          )) OR
    (  _parameterUpdateInternal )  
THEN  
  // reset internal flag for send parameter update
 _parameterUpdateInternal := FALSE;
  // update internal copy of parameters 
 _parCmd := ParCmd;
  // inc parameter sequence
 _command.ParSeq := _command.ParSeq + 1;
  // update command data  
  CommandData := CreateCommandPayload(AxesGroup := AxesGroup); // ( Access via reference to rCommandFB in ACR )
  // notify active command register 
  AxesGroup.Acyclic.ActiveCommandRegister.NotifyParameterChanged := _uniqueID;
  // Reset parameter accepted flag
  ParameterAccepted := FALSE;  
END_IF
END_METHOD

METHOD INTERNAL CreateCommandPayload : RobotLibrarySendDataFB
VAR_IN_OUT
  /// Robot assignment of function
  AxesGroup : AxesGroup; 
END_VAR
// Table 6-547: Sent CMD payload (PLC to RC) of "ReadAnalogInput"
// --------------------------
// Header
// --------------------------
// Byte 00 : UINT  - Type HB     
// Byte 01 :       - Type LB    
// Byte 02 : USINT - Reserve | ExecutionMode
// Byte 03 : USINT - ParSeq  | Priority
// --------------------------
// Datablock
// --------------------------
// Byte 04 : SINT  - EmitterID[0];
// Byte 05 : SINT  - EmitterID[1];
// Byte 06 : SINT  - EmitterID[2];
// Byte 07 : SINT  - EmitterID[3];
// Byte 08 : SINT  - ListenerID;
// Byte 09 : BYTE  - Reserved;
// Byte 10 : USINT - Index;
// --------------------------
// set command parameter 
_command.CmdTyp       :=  CmdType.ReadAnalogInput;
_command.ExecMode     :=  ExecMode;
_command.ParSeq       := _command.ParSeq;
_command.Priority     :=  Priority;
_command.EmitterID[0] := 0;
_command.EmitterID[1] := 0;
_command.EmitterID[2] := 0;
_command.EmitterID[3] := 0;
_command.ListenerID   := _parCmd.ListenerID;
_command.Reserve      := 0;
_command.Index        := _parCmd.Index;


// copy command data to header
_cmdHeader := _command;
// call base implementation to copy header to payload buffer
CreateCommandPayload := SUPER^.CreateCommandPayload(AxesGroup := AxesGroup);

// add command.EmitterID[0]
CreateCommandPayload.AddSint(_command.EmitterID[0]);
// add command.EmitterID[1]
CreateCommandPayload.AddSint(_command.EmitterID[1]);
// add command.EmitterID[2]
CreateCommandPayload.AddSint(_command.EmitterID[2]);
// add command.EmitterID[3]
CreateCommandPayload.AddSint(_command.EmitterID[3]);
// add command.ListenerID
CreateCommandPayload.AddSint(_command.ListenerID);
// add command.Reserve
CreateCommandPayload.AddByte(_command.Reserve);
// add command.Index
CreateCommandPayload.AddUsint(_command.Index);

// Create logging
CreateCommandPayloadLog(AxesGroup := AxesGroup);
END_METHOD

METHOD INTERNAL CreateCommandPayloadLog
VAR_IN_OUT
  /// Robot assignment of function
  AxesGroup : AxesGroup; 
END_VAR
VAR 
  /// internal index for loops
 _idx : DINT;
END_VAR
// Create log entry for Parameter start
CreateLogMessage      ( Timestamp   := AxesGroup.InternalData.SystemTime,
                        MessageType := MessageType.CMD,
                        Severity    := Severity.DEBUG,
                        MessageCode := 0,
                        MessageText := 'Create command payload with the following parameter(s) :');
  
// Create log entry for EmitterID[x]
FOR _idx := 0 TO 3
DO
  CreateLogMessagePara2 ( Timestamp   := AxesGroup.InternalData.SystemTime,
                          MessageType := MessageType.CMD,
                          Severity    := Severity.DEBUG,
                          MessageCode := 0,
                          MessageText := 'Command.EmitterID[{2}] = {1}',
                          Para1       :=  SINT_TO_STRING(_command.EmitterID[_idx]),
                          Para2       :=  DINT_TO_STRING(_idx));
END_FOR

// Create log entry for ListenerID
CreateLogMessagePara1 ( Timestamp   := AxesGroup.InternalData.SystemTime,
                        MessageType := MessageType.CMD,
                        Severity    := Severity.DEBUG,
                        MessageCode := 0,
                        MessageText := 'Command.ListenerID = {1}',
                        Para1       :=  SINT_TO_STRING(_command.ListenerID));
                        
// Create log entry for Reserve
CreateLogMessagePara1 ( Timestamp   := AxesGroup.InternalData.SystemTime,
                        MessageType := MessageType.CMD,
                        Severity    := Severity.DEBUG,
                        MessageCode := 0,
                        MessageText := 'Command.Reserve = {1}',
                        Para1       :=  BYTE_TO_STRING(_command.Reserve));

// Create log entry for Index
CreateLogMessagePara1 ( Timestamp   := AxesGroup.InternalData.SystemTime,
                        MessageType := MessageType.CMD,
                        Severity    := Severity.DEBUG,
                        MessageCode := 0,
                        MessageText := 'Command.Index = {1}',
                        Para1       :=  USINT_TO_STRING(_command.Index));
END_METHOD

METHOD FB_init : BOOL
VAR_INPUT
  /// if TRUE, the retain variables are initialized (warm start / cold start)
  bInitRetains : BOOL; 
  /// if TRUE, the instance afterwards gets moved into the copy code (online change)
  bInCopyCode  : BOOL;  
END_VAR
MyType := 'MC_ReadAnalogInputFB';

ExecMode := ExecutionMode.PARALLEL;
END_METHOD

METHOD PROTECTED OnCall
VAR_IN_OUT
  /// Robot assignment of function
  AxesGroup : AxesGroup; 
END_VAR
// call base implementation
SUPER^.OnCall(AxesGroup := AxesGroup);

CASE _stepCmd OF
  
  00:  IF ( _execute_R.Q )  
       THEN
         // Check function is supported and parameter are valid ?
         IF (( CheckFunctionSupported( AxesGroup := AxesGroup )) AND
             ( CheckParameterValid   ( AxesGroup := AxesGroup )))      
         THEN
           // set busy flag
           Busy := TRUE;
           // Reset command outputs
           SysDepMemSet(pDest := ADR(OutCmd), Value := 0, DataLen := SIZEOF(OutCmd));         
           // apply command parameter
          _parCmd := ParCmd;
           // init parameter sequence
          _command.ParSeq := 1;
           // create command data
           CommandData := CreateCommandPayload(AxesGroup := AxesGroup);
           // Add command to active command register
          _uniqueID := AxesGroup.Acyclic.ActiveCommandRegister.AddCmd( pCommandFB := ADR(THIS^ ));     
           // set timeout
           SetTimeout(PT := _timeoutCmd, rTimer := _timerCmd);
           // inc step counter
          _stepCmd := _stepCmd + 1; 
         END_IF
       END_IF
     

  01:  // Wait for responce received
       IF ( _responseReceived )
       THEN
         // reset response received flag
        _responseReceived := FALSE;

         CASE  _response.State 
         OF
           CmdMessageState.BUFFERED    : CommandBuffered    := TRUE;
           CmdMessageState.ACTIVE      : ParameterAccepted  := TRUE;
           CmdMessageState.INTERRUPTED : CommandInterrupted := TRUE;           
           CmdMessageState.DONE        : Done               := TRUE;
           CmdMessageState.ABORTED     : CommandAborted     := TRUE;
           CmdMessageState.ERROR       : Error              := TRUE;
         END_CASE
                
         // Done, Aborted or Error ?
         IF (_response.State >= CmdMessageState.DONE )            
         THEN
           // Reset Busy flag
           Busy := FALSE;
           // Update results
           OutCmd.OriginID          := _response.OriginID;
           OutCmd.InvocationCounter := _response.InvocationCounter;
           OutCmd.Value             := _response.Value;
           OutCmd.Unit              := _response.Unit;           
           // set timeout
           SetTimeout(PT := _timeoutCmd, rTimer := _timerCmd);
           // inc step counter
          _stepCmd := _stepCmd + 1; 
         END_IF
       END_IF


  02: IF ( NOT Execute)
      THEN
        Reset();
      END_IF
     
ELSE
  // invalid step
  ErrorID := RobotLibraryEvents.ERR_INVALID_STEP;
END_CASE


// Reset FB
IF ( NOT Execute )
THEN
  Reset();
END_IF
END_METHOD

METHOD INTERNAL ParseResponsePayload : DINT
VAR_INPUT
  /// Response data
  ResponseData : RobotLibraryRecvDataFB;
  /// Timestamp
  Timestamp    : SystemTime;  
END_VAR
// Table 6-548: Received CMD payload (RC to PLC) of "ReadAnalogInput"
// --------------------------
// Header
// --------------------------
// Byte 00 : USINT   - ParSeq | State     
// Byte 01 : SINT    - AlarmMessageSeverity    
// Byte 02 : UINT    - AlarmMessageCode HB
// Byte 03 :         - AlarmMessageCode LB
// --------------------------
// Datablock
// --------------------------
// Byte 04 : USINT   - InvocationCounter
// Byte 05 : SINT    - Reserved
// Byte 06 : INT     - Origin ID HB
// Byte 07 : INT       Origin ID LB
// Byte 08 : REAL    - Values HW HB
// Byte 09 :         - Values HW LB
// Byte 10 :         - Values LW HB
// Byte 11 :         - Values LW LB
// Byte 12 : USINT   - Unit
// --------------------------
// call base implementation to parse the header from payload buffer
ResponseData.PayloadPtr := SUPER^.ParseResponsePayload(ResponseData := ResponseData, Timestamp := Timestamp);

// copy parsed header to response
_response.ParSeq               := _rspHeader.ParSeq;
_response.State                := _rspHeader.State;
_response.AlarmMessageSeverity := _rspHeader.AlarmMessageSeverity;
_response.AlarmMessageCode     := _rspHeader.AlarmMessageCode;

// Get Response.InvocationCounter
_response.InvocationCounter := ResponseData.GetUsint();
// Get Response.Reserve
_response.Reserve := ResponseData.GetSint();
// Get Response.OriginID
_response.OriginID := ResponseData.GetInt();
// Get Response.Value
_response.Value := ResponseData.GetReal();
// Get Response.Unit
_response.Unit := ResponseData.GetUsint();

// Create logging
ParseResponsePayloadLog(ResponseData := ResponseData, Timestamp := Timestamp);
END_METHOD

